// TwinCAT 3 PLC project Xplanar_First_Project
// ProgramVersion: 3.1.4023.0
// CompilerDefines: VISU_USEWSTRING
// libraries:
//   cyclic_database_recorder, * (Beckhoff K.K. - Japan)
//   JobManagementFramework, * (Bekchoff Automation K.K.)
//   Tc2_EtherCAT, * (Beckhoff Automation GmbH)
//   Tc2_Standard, * (Beckhoff Automation GmbH)
//   Tc2_System, * (Beckhoff Automation GmbH)
//   Tc2_Utilities, * (Beckhoff Automation GmbH)
//   Tc3_IotBase, * (Beckhoff Automation GmbH)
//   Tc3_JsonXml, * (Beckhoff Automation GmbH)
//   Tc3_Mc3PlanarMotion, * (Beckhoff Automation GmbH)
//   Tc3_Module, * (Beckhoff Automation GmbH)
//   Tc3_Physics, * (Beckhoff Automation GmbH)
//   Tc3_XPlanarUtility, * (Beckhoff Automation GmbH)
//   TwinCATDiagnosisTools, * (Beckhoff Automation K.K.)
//   VisuDialogs, * (System)
//   VisuSymbols,3.5.10.0,System
// project tree:
//   DUTs/ E_DbLogState.TcDUT (not stored), iManualCommand.TcDUT, JobEventReport.TcDUT, ManualCommand.TcDUT, sdo_xplanar_aps_diag.TcDUT, ST_database_aps_diag.TcDUT, ST_database_job_event.TcDUT, ST_mover_dynamics.TcDUT, ST_OperationPanel.TcDUT, ST_RouterStatusInfo.TcDUT, TileInfoType.TcDUT
//   / GlobalTextList.TcGTLO, PlcTask.TcTTO, RecipeManager.TcRMO (not stored), Visualization Manager.TcVMO (not stored)
//   GVLs/ GVL.TcGVL
//   POUs/ IoT.TcPOU, MAIN.TcPOU
//   POUs/model/activities/ FB_TaskMoveA_tilt_Creator.TcPOU, FB_TaskMoveB_tilt.TcPOU, FB_TaskMoveB_tilt_creator.TcPOU, FB_TaskMoveC_creator.TcPOU, FB_TaskMoveToPosition.TcPOU, FB_TaskMoveC.TcPOU, FB_TaskMoveToPosition_creator.TcPOU, FB_TaskMoveZ.TcPOU, FB_TaskMoveA_tilt.TcPOU, FB_TaskMoveZ_creator.TcPOU
//   POUs/model/IoT/ FB_JobReporter.TcPOU, FB_mqtt_publish.TcPOU, FB_serializer.TcPOU
//   VISUs/ ActionMode.TcTLO, MachineMode.TcTLO, Visualization.TcVIS, Visualization_operation.TcVIS, Visualization_recipe.TcVIS
// real-time tasks:
//   TASK Job Task: cycle default, priority 32
//   TASK MC-Task (MET): cycle T#2ms, priority 3, ADS port 521
//   TASK MC-Task (MPT): cycle T#10ms, priority 8, ADS port 531
//   TASK PlcTask: cycle T#10ms, priority 20, ADS port 352
//   TASK XPlanar Task3: cycle T#250us, priority 1, ADS port 350
// I/O:
//   DEVICE Device 3 (EtherCAT), AmsNetId 192.168.80.1.4.1
//     Term 1 (APS4322-7000) [APS4322-7000 Drive]
//       Term 2 (APS4322-5000) [APS4322-5000 Feedback]
//     Term 3 (APS4322-7000) [APS4322-7000 Drive]
//       Term 4 (APS4322-5000) [APS4322-5000 Feedback]
// variable links:
//   Device 3 (EtherCAT) <-> TcCOM Objects/XPlanar/Part1/Tile1
//     Term 3 (APS4322-7000)/APS Comm Inputs/CommStatusWord <-> Data Pointer/MoverCommStatusWord
//     Term 3 (APS4322-7000)/APS Comm Inputs/Data {1..4} <-> Data Pointer/MoverCommDataIn[{0..3}]  (4 links)
//     Term 3 (APS4322-7000)/APS Comm Outputs/CommControlWord <-> Data Pointer/MoverCommControlWord
//     Term 3 (APS4322-7000)/APS Comm Outputs/Data 1 <-> Data Pointer/MoverCommDataOut
//     Term 3 (APS4322-7000)/APS Diagdata/DC Link Voltage <-> Data Pointer/DcLinkVoltage
//     Term 3 (APS4322-7000)/APS Diagdata/Power supply current <-> Data Pointer/PowerSupplyCurrent
//     Term 3 (APS4322-7000)/APS Inputs/StatusWord <-> Data Pointer/PowerUnitStatusWord
//     Term 3 (APS4322-7000)/APS Outputs/ControlWord <-> Data Pointer/PowerUnitControlWord
//     Term 3 (APS4322-7000)/APS Outputs/Current D 0X0 <-> Data Pointer/DCurrentSetPoints[0]
//     Term 3 (APS4322-7000)/APS Outputs/Current D 0X1 <-> Data Pointer/DCurrentSetPoints[1]
//     Term 3 (APS4322-7000)/APS Outputs/Current D 0X2 <-> Data Pointer/DCurrentSetPoints[2]
//     Term 3 (APS4322-7000)/APS Outputs/Current D 1X0 <-> Data Pointer/DCurrentSetPoints[6]
//     Term 3 (APS4322-7000)/APS Outputs/Current D 1X1 <-> Data Pointer/DCurrentSetPoints[7]
//     Term 3 (APS4322-7000)/APS Outputs/Current D 1X2 <-> Data Pointer/DCurrentSetPoints[8]
//     Term 3 (APS4322-7000)/APS Outputs/Current D 2X0 <-> Data Pointer/DCurrentSetPoints[12]
//     Term 3 (APS4322-7000)/APS Outputs/Current D 2X1 <-> Data Pointer/DCurrentSetPoints[13]
//     Term 3 (APS4322-7000)/APS Outputs/Current D 2X2 <-> Data Pointer/DCurrentSetPoints[14]
//     Term 3 (APS4322-7000)/APS Outputs/Current D 3X0 <-> Data Pointer/DCurrentSetPoints[18]
//     Term 3 (APS4322-7000)/APS Outputs/Current D 3X1 <-> Data Pointer/DCurrentSetPoints[19]
//     Term 3 (APS4322-7000)/APS Outputs/Current D 3X2 <-> Data Pointer/DCurrentSetPoints[20]
//     Term 3 (APS4322-7000)/APS Outputs/Current D 0Y0 <-> Data Pointer/DCurrentSetPoints[3]
//     Term 3 (APS4322-7000)/APS Outputs/Current D 0Y1 <-> Data Pointer/DCurrentSetPoints[4]
//     Term 3 (APS4322-7000)/APS Outputs/Current D 0Y2 <-> Data Pointer/DCurrentSetPoints[5]
//     Term 3 (APS4322-7000)/APS Outputs/Current D 1Y0 <-> Data Pointer/DCurrentSetPoints[9]
//     Term 3 (APS4322-7000)/APS Outputs/Current D 1Y1 <-> Data Pointer/DCurrentSetPoints[10]
//     Term 3 (APS4322-7000)/APS Outputs/Current D 1Y2 <-> Data Pointer/DCurrentSetPoints[11]
//     Term 3 (APS4322-7000)/APS Outputs/Current D 2Y0 <-> Data Pointer/DCurrentSetPoints[15]
//     Term 3 (APS4322-7000)/APS Outputs/Current D 2Y1 <-> Data Pointer/DCurrentSetPoints[16]
//     Term 3 (APS4322-7000)/APS Outputs/Current D 2Y2 <-> Data Pointer/DCurrentSetPoints[17]
//     Term 3 (APS4322-7000)/APS Outputs/Current D 3Y0 <-> Data Pointer/DCurrentSetPoints[21]
//     Term 3 (APS4322-7000)/APS Outputs/Current D 3Y1 <-> Data Pointer/DCurrentSetPoints[22]
//     Term 3 (APS4322-7000)/APS Outputs/Current D 3Y2 <-> Data Pointer/DCurrentSetPoints[23]
//     Term 3 (APS4322-7000)/APS Outputs/Current Q 0X0 <-> Data Pointer/QCurrentSetPoints[0]
//     Term 3 (APS4322-7000)/APS Outputs/Current Q 0X1 <-> Data Pointer/QCurrentSetPoints[1]
//     Term 3 (APS4322-7000)/APS Outputs/Current Q 0X2 <-> Data Pointer/QCurrentSetPoints[2]
//     Term 3 (APS4322-7000)/APS Outputs/Current Q 1X0 <-> Data Pointer/QCurrentSetPoints[6]
//     Term 3 (APS4322-7000)/APS Outputs/Current Q 1X1 <-> Data Pointer/QCurrentSetPoints[7]
//     Term 3 (APS4322-7000)/APS Outputs/Current Q 1X2 <-> Data Pointer/QCurrentSetPoints[8]
//     Term 3 (APS4322-7000)/APS Outputs/Current Q 2X0 <-> Data Pointer/QCurrentSetPoints[12]
//     Term 3 (APS4322-7000)/APS Outputs/Current Q 2X1 <-> Data Pointer/QCurrentSetPoints[13]
//     Term 3 (APS4322-7000)/APS Outputs/Current Q 2X2 <-> Data Pointer/QCurrentSetPoints[14]
//     Term 3 (APS4322-7000)/APS Outputs/Current Q 3X0 <-> Data Pointer/QCurrentSetPoints[18]
//     Term 3 (APS4322-7000)/APS Outputs/Current Q 3X1 <-> Data Pointer/QCurrentSetPoints[19]
//     Term 3 (APS4322-7000)/APS Outputs/Current Q 3X2 <-> Data Pointer/QCurrentSetPoints[20]
//     Term 3 (APS4322-7000)/APS Outputs/Current Q 0Y0 <-> Data Pointer/QCurrentSetPoints[3]
//     Term 3 (APS4322-7000)/APS Outputs/Current Q 0Y1 <-> Data Pointer/QCurrentSetPoints[4]
//     Term 3 (APS4322-7000)/APS Outputs/Current Q 0Y2 <-> Data Pointer/QCurrentSetPoints[5]
//     Term 3 (APS4322-7000)/APS Outputs/Current Q 1Y0 <-> Data Pointer/QCurrentSetPoints[9]
//     Term 3 (APS4322-7000)/APS Outputs/Current Q 1Y1 <-> Data Pointer/QCurrentSetPoints[10]
//     Term 3 (APS4322-7000)/APS Outputs/Current Q 1Y2 <-> Data Pointer/QCurrentSetPoints[11]
//     Term 3 (APS4322-7000)/APS Outputs/Current Q 2Y0 <-> Data Pointer/QCurrentSetPoints[15]
//     Term 3 (APS4322-7000)/APS Outputs/Current Q 2Y1 <-> Data Pointer/QCurrentSetPoints[16]
//     Term 3 (APS4322-7000)/APS Outputs/Current Q 2Y2 <-> Data Pointer/QCurrentSetPoints[17]
//     Term 3 (APS4322-7000)/APS Outputs/Current Q 3Y0 <-> Data Pointer/QCurrentSetPoints[21]
//     Term 3 (APS4322-7000)/APS Outputs/Current Q 3Y1 <-> Data Pointer/QCurrentSetPoints[22]
//     Term 3 (APS4322-7000)/APS Outputs/Current Q 3Y2 <-> Data Pointer/QCurrentSetPoints[23]
//     Term 3 (APS4322-7000)/APS Outputs/PhiE 0X0 <-> Data Pointer/PhiSetPoints[0]
//     Term 3 (APS4322-7000)/APS Outputs/PhiE 0X1 <-> Data Pointer/PhiSetPoints[1]
//     Term 3 (APS4322-7000)/APS Outputs/PhiE 0X2 <-> Data Pointer/PhiSetPoints[2]
//     Term 3 (APS4322-7000)/APS Outputs/PhiE 1X0 <-> Data Pointer/PhiSetPoints[6]
//     Term 3 (APS4322-7000)/APS Outputs/PhiE 1X1 <-> Data Pointer/PhiSetPoints[7]
//     Term 3 (APS4322-7000)/APS Outputs/PhiE 1X2 <-> Data Pointer/PhiSetPoints[8]
//     Term 3 (APS4322-7000)/APS Outputs/PhiE 2X0 <-> Data Pointer/PhiSetPoints[12]
//     Term 3 (APS4322-7000)/APS Outputs/PhiE 2X1 <-> Data Pointer/PhiSetPoints[13]
//     Term 3 (APS4322-7000)/APS Outputs/PhiE 2X2 <-> Data Pointer/PhiSetPoints[14]
//     Term 3 (APS4322-7000)/APS Outputs/PhiE 3X0 <-> Data Pointer/PhiSetPoints[18]
//     Term 3 (APS4322-7000)/APS Outputs/PhiE 3X1 <-> Data Pointer/PhiSetPoints[19]
//     Term 3 (APS4322-7000)/APS Outputs/PhiE 3X2 <-> Data Pointer/PhiSetPoints[20]
//     Term 3 (APS4322-7000)/APS Outputs/PhiE 0Y0 <-> Data Pointer/PhiSetPoints[3]
//     Term 3 (APS4322-7000)/APS Outputs/PhiE 0Y1 <-> Data Pointer/PhiSetPoints[4]
//     Term 3 (APS4322-7000)/APS Outputs/PhiE 0Y2 <-> Data Pointer/PhiSetPoints[5]
//     Term 3 (APS4322-7000)/APS Outputs/PhiE 1Y0 <-> Data Pointer/PhiSetPoints[9]
//     Term 3 (APS4322-7000)/APS Outputs/PhiE 1Y1 <-> Data Pointer/PhiSetPoints[10]
//     Term 3 (APS4322-7000)/APS Outputs/PhiE 1Y2 <-> Data Pointer/PhiSetPoints[11]
//     Term 3 (APS4322-7000)/APS Outputs/PhiE 2Y0 <-> Data Pointer/PhiSetPoints[15]
//     Term 3 (APS4322-7000)/APS Outputs/PhiE 2Y1 <-> Data Pointer/PhiSetPoints[16]
//     Term 3 (APS4322-7000)/APS Outputs/PhiE 2Y2 <-> Data Pointer/PhiSetPoints[17]
//     Term 3 (APS4322-7000)/APS Outputs/PhiE 3Y0 <-> Data Pointer/PhiSetPoints[21]
//     Term 3 (APS4322-7000)/APS Outputs/PhiE 3Y1 <-> Data Pointer/PhiSetPoints[22]
//     Term 3 (APS4322-7000)/APS Outputs/PhiE 3Y2 <-> Data Pointer/PhiSetPoints[23]
//     Term 3 (APS4322-7000)/Term 4 (APS4322-5000)/FB Inputs/A{0..8 step 2} X-Field <-> Data Pointer/HallSensorFieldsXYZ[{0..12 step 3}]  (5 links)
//     Term 3 (APS4322-7000)/Term 4 (APS4322-5000)/FB Inputs/A{0..8 step 2} Y-Field <-> Data Pointer/HallSensorFieldsXYZ[{1..13 step 3}]  (5 links)
//     Term 3 (APS4322-7000)/Term 4 (APS4322-5000)/FB Inputs/A{0..8 step 2} Z-Field <-> Data Pointer/HallSensorFieldsXYZ[{2..14 step 3}]  (5 links)
//     Term 3 (APS4322-7000)/Term 4 (APS4322-5000)/FB Inputs/B{1..9 step 2} X-Field <-> Data Pointer/HallSensorFieldsXYZ[{15..27 step 3}]  (5 links)
//     Term 3 (APS4322-7000)/Term 4 (APS4322-5000)/FB Inputs/B{1..9 step 2} Y-Field <-> Data Pointer/HallSensorFieldsXYZ[{16..28 step 3}]  (5 links)
//     Term 3 (APS4322-7000)/Term 4 (APS4322-5000)/FB Inputs/B{1..9 step 2} Z-Field <-> Data Pointer/HallSensorFieldsXYZ[{17..29 step 3}]  (5 links)
//     Term 3 (APS4322-7000)/Term 4 (APS4322-5000)/FB Inputs/C{0..8 step 2} X-Field <-> Data Pointer/HallSensorFieldsXYZ[{30..42 step 3}]  (5 links)
//     Term 3 (APS4322-7000)/Term 4 (APS4322-5000)/FB Inputs/C{0..8 step 2} Y-Field <-> Data Pointer/HallSensorFieldsXYZ[{31..43 step 3}]  (5 links)
//     Term 3 (APS4322-7000)/Term 4 (APS4322-5000)/FB Inputs/C{0..8 step 2} Z-Field <-> Data Pointer/HallSensorFieldsXYZ[{32..44 step 3}]  (5 links)
//     Term 3 (APS4322-7000)/Term 4 (APS4322-5000)/FB Inputs/D{1..9 step 2} X-Field <-> Data Pointer/HallSensorFieldsXYZ[{45..57 step 3}]  (5 links)
//     Term 3 (APS4322-7000)/Term 4 (APS4322-5000)/FB Inputs/D{1..9 step 2} Y-Field <-> Data Pointer/HallSensorFieldsXYZ[{46..58 step 3}]  (5 links)
//     Term 3 (APS4322-7000)/Term 4 (APS4322-5000)/FB Inputs/D{1..9 step 2} Z-Field <-> Data Pointer/HallSensorFieldsXYZ[{47..59 step 3}]  (5 links)
//     Term 3 (APS4322-7000)/Term 4 (APS4322-5000)/FB Inputs/E{0..8 step 2} X-Field <-> Data Pointer/HallSensorFieldsXYZ[{60..72 step 3}]  (5 links)
//     Term 3 (APS4322-7000)/Term 4 (APS4322-5000)/FB Inputs/E{0..8 step 2} Y-Field <-> Data Pointer/HallSensorFieldsXYZ[{61..73 step 3}]  (5 links)
//     Term 3 (APS4322-7000)/Term 4 (APS4322-5000)/FB Inputs/E{0..8 step 2} Z-Field <-> Data Pointer/HallSensorFieldsXYZ[{62..74 step 3}]  (5 links)
//     Term 3 (APS4322-7000)/Term 4 (APS4322-5000)/FB Inputs/F{1..9 step 2} X-Field <-> Data Pointer/HallSensorFieldsXYZ[{75..87 step 3}]  (5 links)
//     Term 3 (APS4322-7000)/Term 4 (APS4322-5000)/FB Inputs/F{1..9 step 2} Y-Field <-> Data Pointer/HallSensorFieldsXYZ[{76..88 step 3}]  (5 links)
//     Term 3 (APS4322-7000)/Term 4 (APS4322-5000)/FB Inputs/F{1..9 step 2} Z-Field <-> Data Pointer/HallSensorFieldsXYZ[{77..89 step 3}]  (5 links)
//     Term 3 (APS4322-7000)/Term 4 (APS4322-5000)/FB Inputs/G{0..8 step 2} X-Field <-> Data Pointer/HallSensorFieldsXYZ[{90..102 step 3}]  (5 links)
//     Term 3 (APS4322-7000)/Term 4 (APS4322-5000)/FB Inputs/G{0..8 step 2} Y-Field <-> Data Pointer/HallSensorFieldsXYZ[{91..103 step 3}]  (5 links)
//     Term 3 (APS4322-7000)/Term 4 (APS4322-5000)/FB Inputs/G{0..8 step 2} Z-Field <-> Data Pointer/HallSensorFieldsXYZ[{92..104 step 3}]  (5 links)
//     Term 3 (APS4322-7000)/Term 4 (APS4322-5000)/FB Inputs/H{1..9 step 2} X-Field <-> Data Pointer/HallSensorFieldsXYZ[{105..117 step 3}]  (5 links)
//     Term 3 (APS4322-7000)/Term 4 (APS4322-5000)/FB Inputs/H{1..9 step 2} Y-Field <-> Data Pointer/HallSensorFieldsXYZ[{106..118 step 3}]  (5 links)
//     Term 3 (APS4322-7000)/Term 4 (APS4322-5000)/FB Inputs/H{1..9 step 2} Z-Field <-> Data Pointer/HallSensorFieldsXYZ[{107..119 step 3}]  (5 links)
//     Term 3 (APS4322-7000)/Term 4 (APS4322-5000)/FB Inputs/I{0..8 step 2} X-Field <-> Data Pointer/HallSensorFieldsXYZ[{120..132 step 3}]  (5 links)
//     Term 3 (APS4322-7000)/Term 4 (APS4322-5000)/FB Inputs/I{0..8 step 2} Y-Field <-> Data Pointer/HallSensorFieldsXYZ[{121..133 step 3}]  (5 links)
//     Term 3 (APS4322-7000)/Term 4 (APS4322-5000)/FB Inputs/I{0..8 step 2} Z-Field <-> Data Pointer/HallSensorFieldsXYZ[{122..134 step 3}]  (5 links)
//     Term 3 (APS4322-7000)/Term 4 (APS4322-5000)/FB Inputs/J{1..9 step 2} X-Field <-> Data Pointer/HallSensorFieldsXYZ[{135..147 step 3}]  (5 links)
//     Term 3 (APS4322-7000)/Term 4 (APS4322-5000)/FB Inputs/J{1..9 step 2} Y-Field <-> Data Pointer/HallSensorFieldsXYZ[{136..148 step 3}]  (5 links)
//     Term 3 (APS4322-7000)/Term 4 (APS4322-5000)/FB Inputs/J{1..9 step 2} Z-Field <-> Data Pointer/HallSensorFieldsXYZ[{137..149 step 3}]  (5 links)
//     Term 3 (APS4322-7000)/Term 4 (APS4322-5000)/FB Inputs/Status <-> Data Pointer/FeedbackStatus
//   Device 3 (EtherCAT) <-> TcCOM Objects/XPlanar/Part1/Tile2
//     Term 1 (APS4322-7000)/APS Comm Inputs/CommStatusWord <-> Data Pointer/MoverCommStatusWord
//     Term 1 (APS4322-7000)/APS Comm Inputs/Data {1..4} <-> Data Pointer/MoverCommDataIn[{0..3}]  (4 links)
//     Term 1 (APS4322-7000)/APS Comm Outputs/CommControlWord <-> Data Pointer/MoverCommControlWord
//     Term 1 (APS4322-7000)/APS Comm Outputs/Data 1 <-> Data Pointer/MoverCommDataOut
//     Term 1 (APS4322-7000)/APS Diagdata/DC Link Voltage <-> Data Pointer/DcLinkVoltage
//     Term 1 (APS4322-7000)/APS Diagdata/Power supply current <-> Data Pointer/PowerSupplyCurrent
//     Term 1 (APS4322-7000)/APS Inputs/StatusWord <-> Data Pointer/PowerUnitStatusWord
//     Term 1 (APS4322-7000)/APS Outputs/ControlWord <-> Data Pointer/PowerUnitControlWord
//     Term 1 (APS4322-7000)/APS Outputs/Current D 0X0 <-> Data Pointer/DCurrentSetPoints[0]
//     Term 1 (APS4322-7000)/APS Outputs/Current D 0X1 <-> Data Pointer/DCurrentSetPoints[1]
//     Term 1 (APS4322-7000)/APS Outputs/Current D 0X2 <-> Data Pointer/DCurrentSetPoints[2]
//     Term 1 (APS4322-7000)/APS Outputs/Current D 1X0 <-> Data Pointer/DCurrentSetPoints[6]
//     Term 1 (APS4322-7000)/APS Outputs/Current D 1X1 <-> Data Pointer/DCurrentSetPoints[7]
//     Term 1 (APS4322-7000)/APS Outputs/Current D 1X2 <-> Data Pointer/DCurrentSetPoints[8]
//     Term 1 (APS4322-7000)/APS Outputs/Current D 2X0 <-> Data Pointer/DCurrentSetPoints[12]
//     Term 1 (APS4322-7000)/APS Outputs/Current D 2X1 <-> Data Pointer/DCurrentSetPoints[13]
//     Term 1 (APS4322-7000)/APS Outputs/Current D 2X2 <-> Data Pointer/DCurrentSetPoints[14]
//     Term 1 (APS4322-7000)/APS Outputs/Current D 3X0 <-> Data Pointer/DCurrentSetPoints[18]
//     Term 1 (APS4322-7000)/APS Outputs/Current D 3X1 <-> Data Pointer/DCurrentSetPoints[19]
//     Term 1 (APS4322-7000)/APS Outputs/Current D 3X2 <-> Data Pointer/DCurrentSetPoints[20]
//     Term 1 (APS4322-7000)/APS Outputs/Current D 0Y0 <-> Data Pointer/DCurrentSetPoints[3]
//     Term 1 (APS4322-7000)/APS Outputs/Current D 0Y1 <-> Data Pointer/DCurrentSetPoints[4]
//     Term 1 (APS4322-7000)/APS Outputs/Current D 0Y2 <-> Data Pointer/DCurrentSetPoints[5]
//     Term 1 (APS4322-7000)/APS Outputs/Current D 1Y0 <-> Data Pointer/DCurrentSetPoints[9]
//     Term 1 (APS4322-7000)/APS Outputs/Current D 1Y1 <-> Data Pointer/DCurrentSetPoints[10]
//     Term 1 (APS4322-7000)/APS Outputs/Current D 1Y2 <-> Data Pointer/DCurrentSetPoints[11]
//     Term 1 (APS4322-7000)/APS Outputs/Current D 2Y0 <-> Data Pointer/DCurrentSetPoints[15]
//     Term 1 (APS4322-7000)/APS Outputs/Current D 2Y1 <-> Data Pointer/DCurrentSetPoints[16]
//     Term 1 (APS4322-7000)/APS Outputs/Current D 2Y2 <-> Data Pointer/DCurrentSetPoints[17]
//     Term 1 (APS4322-7000)/APS Outputs/Current D 3Y0 <-> Data Pointer/DCurrentSetPoints[21]
//     Term 1 (APS4322-7000)/APS Outputs/Current D 3Y1 <-> Data Pointer/DCurrentSetPoints[22]
//     Term 1 (APS4322-7000)/APS Outputs/Current D 3Y2 <-> Data Pointer/DCurrentSetPoints[23]
//     Term 1 (APS4322-7000)/APS Outputs/Current Q 0X0 <-> Data Pointer/QCurrentSetPoints[0]
//     Term 1 (APS4322-7000)/APS Outputs/Current Q 0X1 <-> Data Pointer/QCurrentSetPoints[1]
//     Term 1 (APS4322-7000)/APS Outputs/Current Q 0X2 <-> Data Pointer/QCurrentSetPoints[2]
//     Term 1 (APS4322-7000)/APS Outputs/Current Q 1X0 <-> Data Pointer/QCurrentSetPoints[6]
//     Term 1 (APS4322-7000)/APS Outputs/Current Q 1X1 <-> Data Pointer/QCurrentSetPoints[7]
//     Term 1 (APS4322-7000)/APS Outputs/Current Q 1X2 <-> Data Pointer/QCurrentSetPoints[8]
//     Term 1 (APS4322-7000)/APS Outputs/Current Q 2X0 <-> Data Pointer/QCurrentSetPoints[12]
//     Term 1 (APS4322-7000)/APS Outputs/Current Q 2X1 <-> Data Pointer/QCurrentSetPoints[13]
//     Term 1 (APS4322-7000)/APS Outputs/Current Q 2X2 <-> Data Pointer/QCurrentSetPoints[14]
//     Term 1 (APS4322-7000)/APS Outputs/Current Q 3X0 <-> Data Pointer/QCurrentSetPoints[18]
//     Term 1 (APS4322-7000)/APS Outputs/Current Q 3X1 <-> Data Pointer/QCurrentSetPoints[19]
//     Term 1 (APS4322-7000)/APS Outputs/Current Q 3X2 <-> Data Pointer/QCurrentSetPoints[20]
//     Term 1 (APS4322-7000)/APS Outputs/Current Q 0Y0 <-> Data Pointer/QCurrentSetPoints[3]
//     Term 1 (APS4322-7000)/APS Outputs/Current Q 0Y1 <-> Data Pointer/QCurrentSetPoints[4]
//     Term 1 (APS4322-7000)/APS Outputs/Current Q 0Y2 <-> Data Pointer/QCurrentSetPoints[5]
//     Term 1 (APS4322-7000)/APS Outputs/Current Q 1Y0 <-> Data Pointer/QCurrentSetPoints[9]
//     Term 1 (APS4322-7000)/APS Outputs/Current Q 1Y1 <-> Data Pointer/QCurrentSetPoints[10]
//     Term 1 (APS4322-7000)/APS Outputs/Current Q 1Y2 <-> Data Pointer/QCurrentSetPoints[11]
//     Term 1 (APS4322-7000)/APS Outputs/Current Q 2Y0 <-> Data Pointer/QCurrentSetPoints[15]
//     Term 1 (APS4322-7000)/APS Outputs/Current Q 2Y1 <-> Data Pointer/QCurrentSetPoints[16]
//     Term 1 (APS4322-7000)/APS Outputs/Current Q 2Y2 <-> Data Pointer/QCurrentSetPoints[17]
//     Term 1 (APS4322-7000)/APS Outputs/Current Q 3Y0 <-> Data Pointer/QCurrentSetPoints[21]
//     Term 1 (APS4322-7000)/APS Outputs/Current Q 3Y1 <-> Data Pointer/QCurrentSetPoints[22]
//     Term 1 (APS4322-7000)/APS Outputs/Current Q 3Y2 <-> Data Pointer/QCurrentSetPoints[23]
//     Term 1 (APS4322-7000)/APS Outputs/PhiE 0X0 <-> Data Pointer/PhiSetPoints[0]
//     Term 1 (APS4322-7000)/APS Outputs/PhiE 0X1 <-> Data Pointer/PhiSetPoints[1]
//     Term 1 (APS4322-7000)/APS Outputs/PhiE 0X2 <-> Data Pointer/PhiSetPoints[2]
//     Term 1 (APS4322-7000)/APS Outputs/PhiE 1X0 <-> Data Pointer/PhiSetPoints[6]
//     Term 1 (APS4322-7000)/APS Outputs/PhiE 1X1 <-> Data Pointer/PhiSetPoints[7]
//     Term 1 (APS4322-7000)/APS Outputs/PhiE 1X2 <-> Data Pointer/PhiSetPoints[8]
//     Term 1 (APS4322-7000)/APS Outputs/PhiE 2X0 <-> Data Pointer/PhiSetPoints[12]
//     Term 1 (APS4322-7000)/APS Outputs/PhiE 2X1 <-> Data Pointer/PhiSetPoints[13]
//     Term 1 (APS4322-7000)/APS Outputs/PhiE 2X2 <-> Data Pointer/PhiSetPoints[14]
//     Term 1 (APS4322-7000)/APS Outputs/PhiE 3X0 <-> Data Pointer/PhiSetPoints[18]
//     Term 1 (APS4322-7000)/APS Outputs/PhiE 3X1 <-> Data Pointer/PhiSetPoints[19]
//     Term 1 (APS4322-7000)/APS Outputs/PhiE 3X2 <-> Data Pointer/PhiSetPoints[20]
//     Term 1 (APS4322-7000)/APS Outputs/PhiE 0Y0 <-> Data Pointer/PhiSetPoints[3]
//     Term 1 (APS4322-7000)/APS Outputs/PhiE 0Y1 <-> Data Pointer/PhiSetPoints[4]
//     Term 1 (APS4322-7000)/APS Outputs/PhiE 0Y2 <-> Data Pointer/PhiSetPoints[5]
//     Term 1 (APS4322-7000)/APS Outputs/PhiE 1Y0 <-> Data Pointer/PhiSetPoints[9]
//     Term 1 (APS4322-7000)/APS Outputs/PhiE 1Y1 <-> Data Pointer/PhiSetPoints[10]
//     Term 1 (APS4322-7000)/APS Outputs/PhiE 1Y2 <-> Data Pointer/PhiSetPoints[11]
//     Term 1 (APS4322-7000)/APS Outputs/PhiE 2Y0 <-> Data Pointer/PhiSetPoints[15]
//     Term 1 (APS4322-7000)/APS Outputs/PhiE 2Y1 <-> Data Pointer/PhiSetPoints[16]
//     Term 1 (APS4322-7000)/APS Outputs/PhiE 2Y2 <-> Data Pointer/PhiSetPoints[17]
//     Term 1 (APS4322-7000)/APS Outputs/PhiE 3Y0 <-> Data Pointer/PhiSetPoints[21]
//     Term 1 (APS4322-7000)/APS Outputs/PhiE 3Y1 <-> Data Pointer/PhiSetPoints[22]
//     Term 1 (APS4322-7000)/APS Outputs/PhiE 3Y2 <-> Data Pointer/PhiSetPoints[23]
//     Term 1 (APS4322-7000)/Term 2 (APS4322-5000)/FB Inputs/A{0..8 step 2} X-Field <-> Data Pointer/HallSensorFieldsXYZ[{0..12 step 3}]  (5 links)
//     Term 1 (APS4322-7000)/Term 2 (APS4322-5000)/FB Inputs/A{0..8 step 2} Y-Field <-> Data Pointer/HallSensorFieldsXYZ[{1..13 step 3}]  (5 links)
//     Term 1 (APS4322-7000)/Term 2 (APS4322-5000)/FB Inputs/A{0..8 step 2} Z-Field <-> Data Pointer/HallSensorFieldsXYZ[{2..14 step 3}]  (5 links)
//     Term 1 (APS4322-7000)/Term 2 (APS4322-5000)/FB Inputs/B{1..9 step 2} X-Field <-> Data Pointer/HallSensorFieldsXYZ[{15..27 step 3}]  (5 links)
//     Term 1 (APS4322-7000)/Term 2 (APS4322-5000)/FB Inputs/B{1..9 step 2} Y-Field <-> Data Pointer/HallSensorFieldsXYZ[{16..28 step 3}]  (5 links)
//     Term 1 (APS4322-7000)/Term 2 (APS4322-5000)/FB Inputs/B{1..9 step 2} Z-Field <-> Data Pointer/HallSensorFieldsXYZ[{17..29 step 3}]  (5 links)
//     Term 1 (APS4322-7000)/Term 2 (APS4322-5000)/FB Inputs/C{0..8 step 2} X-Field <-> Data Pointer/HallSensorFieldsXYZ[{30..42 step 3}]  (5 links)
//     Term 1 (APS4322-7000)/Term 2 (APS4322-5000)/FB Inputs/C{0..8 step 2} Y-Field <-> Data Pointer/HallSensorFieldsXYZ[{31..43 step 3}]  (5 links)
//     Term 1 (APS4322-7000)/Term 2 (APS4322-5000)/FB Inputs/C{0..8 step 2} Z-Field <-> Data Pointer/HallSensorFieldsXYZ[{32..44 step 3}]  (5 links)
//     Term 1 (APS4322-7000)/Term 2 (APS4322-5000)/FB Inputs/D{1..9 step 2} X-Field <-> Data Pointer/HallSensorFieldsXYZ[{45..57 step 3}]  (5 links)
//     Term 1 (APS4322-7000)/Term 2 (APS4322-5000)/FB Inputs/D{1..9 step 2} Y-Field <-> Data Pointer/HallSensorFieldsXYZ[{46..58 step 3}]  (5 links)
//     Term 1 (APS4322-7000)/Term 2 (APS4322-5000)/FB Inputs/D{1..9 step 2} Z-Field <-> Data Pointer/HallSensorFieldsXYZ[{47..59 step 3}]  (5 links)
//     Term 1 (APS4322-7000)/Term 2 (APS4322-5000)/FB Inputs/E{0..8 step 2} X-Field <-> Data Pointer/HallSensorFieldsXYZ[{60..72 step 3}]  (5 links)
//     Term 1 (APS4322-7000)/Term 2 (APS4322-5000)/FB Inputs/E{0..8 step 2} Y-Field <-> Data Pointer/HallSensorFieldsXYZ[{61..73 step 3}]  (5 links)
//     Term 1 (APS4322-7000)/Term 2 (APS4322-5000)/FB Inputs/E{0..8 step 2} Z-Field <-> Data Pointer/HallSensorFieldsXYZ[{62..74 step 3}]  (5 links)
//     Term 1 (APS4322-7000)/Term 2 (APS4322-5000)/FB Inputs/F{1..9 step 2} X-Field <-> Data Pointer/HallSensorFieldsXYZ[{75..87 step 3}]  (5 links)
//     Term 1 (APS4322-7000)/Term 2 (APS4322-5000)/FB Inputs/F{1..9 step 2} Y-Field <-> Data Pointer/HallSensorFieldsXYZ[{76..88 step 3}]  (5 links)
//     Term 1 (APS4322-7000)/Term 2 (APS4322-5000)/FB Inputs/F{1..9 step 2} Z-Field <-> Data Pointer/HallSensorFieldsXYZ[{77..89 step 3}]  (5 links)
//     Term 1 (APS4322-7000)/Term 2 (APS4322-5000)/FB Inputs/G{0..8 step 2} X-Field <-> Data Pointer/HallSensorFieldsXYZ[{90..102 step 3}]  (5 links)
//     Term 1 (APS4322-7000)/Term 2 (APS4322-5000)/FB Inputs/G{0..8 step 2} Y-Field <-> Data Pointer/HallSensorFieldsXYZ[{91..103 step 3}]  (5 links)
//     Term 1 (APS4322-7000)/Term 2 (APS4322-5000)/FB Inputs/G{0..8 step 2} Z-Field <-> Data Pointer/HallSensorFieldsXYZ[{92..104 step 3}]  (5 links)
//     Term 1 (APS4322-7000)/Term 2 (APS4322-5000)/FB Inputs/H{1..9 step 2} X-Field <-> Data Pointer/HallSensorFieldsXYZ[{105..117 step 3}]  (5 links)
//     Term 1 (APS4322-7000)/Term 2 (APS4322-5000)/FB Inputs/H{1..9 step 2} Y-Field <-> Data Pointer/HallSensorFieldsXYZ[{106..118 step 3}]  (5 links)
//     Term 1 (APS4322-7000)/Term 2 (APS4322-5000)/FB Inputs/H{1..9 step 2} Z-Field <-> Data Pointer/HallSensorFieldsXYZ[{107..119 step 3}]  (5 links)
//     Term 1 (APS4322-7000)/Term 2 (APS4322-5000)/FB Inputs/I{0..8 step 2} X-Field <-> Data Pointer/HallSensorFieldsXYZ[{120..132 step 3}]  (5 links)
//     Term 1 (APS4322-7000)/Term 2 (APS4322-5000)/FB Inputs/I{0..8 step 2} Y-Field <-> Data Pointer/HallSensorFieldsXYZ[{121..133 step 3}]  (5 links)
//     Term 1 (APS4322-7000)/Term 2 (APS4322-5000)/FB Inputs/I{0..8 step 2} Z-Field <-> Data Pointer/HallSensorFieldsXYZ[{122..134 step 3}]  (5 links)
//     Term 1 (APS4322-7000)/Term 2 (APS4322-5000)/FB Inputs/J{1..9 step 2} X-Field <-> Data Pointer/HallSensorFieldsXYZ[{135..147 step 3}]  (5 links)
//     Term 1 (APS4322-7000)/Term 2 (APS4322-5000)/FB Inputs/J{1..9 step 2} Y-Field <-> Data Pointer/HallSensorFieldsXYZ[{136..148 step 3}]  (5 links)
//     Term 1 (APS4322-7000)/Term 2 (APS4322-5000)/FB Inputs/J{1..9 step 2} Z-Field <-> Data Pointer/HallSensorFieldsXYZ[{137..149 step 3}]  (5 links)
//     Term 1 (APS4322-7000)/Term 2 (APS4322-5000)/FB Inputs/Status <-> Data Pointer/FeedbackStatus
//   XPlanar MC Project/Axes/Mover4220_1 <-> TcCOM Objects/XPlanar/Mover4220_1
//     McToIo/STD <-> InputsFromNC3/NC3ToHW
//   Xplanar_First_Project/Xplanar_First_Project Instance <-> XPlanar MC Project/Axes/Mover4220_1
//     PlcTask Inputs/GVL.planar_movers[1].MCTOPLC/ACT <-> McToPlc/ACT
//     PlcTask Inputs/GVL.planar_movers[1].MCTOPLC/COORDMODE <-> McToPlc/COORDMODE
//     PlcTask Inputs/GVL.planar_movers[1].MCTOPLC/SET <-> McToPlc/SET
//     PlcTask Inputs/GVL.planar_movers[1].MCTOPLC/SETONTRACK <-> McToPlc/SETONTRACK
//     PlcTask Inputs/GVL.planar_movers[1].MCTOPLC/STD <-> McToPlc/STD
//     PlcTask Outputs/GVL.planar_movers[1].PLCTOMC/STD <-> PlcToMc/STD
//   TcCOM Objects/XPlanar/Mover4220_1 <-> XPlanar MC Project/Axes/Mover4220_1
//     OutputsToNC3/HWToNC3 <-> IoToMc/STD

CONFIGURATION Xplanar_First_Project
    RESOURCE PLC ON TwinCAT3
        TASK PlcTask(INTERVAL := T#10ms, PRIORITY := 20);
        PROGRAM MAIN WITH PlcTask : MAIN;
    END_RESOURCE
END_CONFIGURATION

// ---- DUTs/iManualCommand.TcDUT
TYPE iManualCommand :
UNION
	i_com: UINT;
	com: ManualCommand;
END_UNION
END_TYPE

// ---- DUTs/JobEventReport.TcDUT
{attribute ‘pack_mode’ := ‘1’}
TYPE JobEventReport :
STRUCT
	old_state	: STRING;
	new_state	: STRING;
	record_time	: STRING;
	{attribute 'TcEncoding':='UTF-8'}
	job_id		: STRING;
	{attribute 'TcEncoding':='UTF-8'}
	task_name	: STRING;
	erro_id		: UDINT;
END_STRUCT
END_TYPE

// ---- DUTs/ManualCommand.TcDUT
{attribute 'qualified_only'}
{attribute 'strict'}
TYPE ManualCommand :
(
	move_pos_L1 := 0,
	move_pos_L2,
	move_pos_L3,
	move_pos_c1,
	move_pos_c2,
	move_pos_c3,
	move_pos_r1,
	move_pos_r2,
	move_pos_r3,
	move_up,
	move_down,
	move_tilt_up_front,
	move_tilt_up_rear,
	move_tilt_up_right,
	move_tilt_up_left,
	move_tilt_horizontal,
	move_roll_w,
	move_roll_n,
	move_roll_e,
	move_roll_s
);
END_TYPE

// ---- DUTs/sdo_xplanar_aps_diag.TcDUT
{attribute 'TcAnalytics'}
{attribute 'pack_mode' := '4'}
TYPE sdo_xplanar_aps_diag :
STRUCT
  identity: USINT;
  {attribute 'FieldName' := 'dc_link_voltage'}
  dc_link_voltage: DINT;
  {attribute 'FieldName' := 'power_supply_current'}
  power_supply_current: DINT;
  {attribute 'FieldName' := 'temperature_north'}
  temperature_north: UINT;
  {attribute 'FieldName' := 'temperature_east'}
  temperature_east: UINT;
  {attribute 'FieldName' := 'temperature_south'}
  temperature_south: UINT;
  {attribute 'FieldName' := 'temperature_west'}
  temperature_west: UINT;
  {attribute 'FieldName' := 'temperature_center'}
  temperature_center: UINT;
  {attribute 'FieldName' := 'temperature_power'}
  temperature_power: UINT;
  {attribute 'FieldName' := 'fan_rpm'}
  fan_rpm: UINT;
  {attribute 'FieldName' := 'fan_duty_cycle'}
  fan_duty_cycle: USINT;
  {attribute 'FieldName' := 'supply_voltage_us'}
  supply_voltage_us: UDINT;
  {attribute 'FieldName' := 'auxiliary_voltage'}
  auxiliary_voltage: UDINT;
  {attribute 'FieldName' := 'acceleration_x'}
  acceleration_x: UDINT;
  {attribute 'FieldName' := 'acceleration_y'}
  acceleration_y: UDINT;
  {attribute 'FieldName' := 'acceleration_z'}
  acceleration_z: UDINT;
  {attribute 'FieldName' := 'time_to_shutdown'}
  time_to_shutdown: UDINT;
  {attribute 'FieldName' := 'fb_fw_rev'}
  fb_fw_rev: UDINT;
END_STRUCT
END_TYPE

// ---- DUTs/ST_database_aps_diag.TcDUT
{attribute 'pack_mode' := '1'}
TYPE ST_database_aps_diag:
STRUCT
	{attribute 'TagName' := 'tile_number'}
	tile_number :STRING;
	{attribute 'FieldName' := 'dc_link_voltage'}
	dc_link_voltage: DINT;
	{attribute 'FieldName' := 'power_supply_current'}
	power_supply_current: DINT;
	{attribute 'FieldName' := 'temperature_north'}
	temperature_north: DINT;
	{attribute 'FieldName' := 'temperature_east'}
	temperature_east: DINT;
	{attribute 'FieldName' := 'temperature_south'}
	temperature_south: DINT;
	{attribute 'FieldName' := 'temperature_west'}
	temperature_west: DINT;
	{attribute 'FieldName' := 'temperature_center'}
	temperature_center: DINT;
	{attribute 'FieldName' := 'temperature_power'}
	temperature_power: DINT;
	{attribute 'FieldName' := 'fan_rpm'}
	fan_rpm: DINT;
	{attribute 'FieldName' := 'fan_duty_cycle'}
	fan_duty_cycle: INT;
	{attribute 'FieldName' := 'supply_voltage_us'}
	supply_voltage_us: LINT;
	{attribute 'FieldName' := 'auxiliary_voltage'}
	auxiliary_voltage: LINT;
	{attribute 'FieldName' := 'acceleration_x'}
	acceleration_x: LINT;
	{attribute 'FieldName' := 'acceleration_y'}
	acceleration_y: LINT;
	{attribute 'FieldName' := 'acceleration_z'}
	acceleration_z: LINT;
	{attribute 'FieldName' := 'time_to_shutdown'}
	time_to_shutdown: LINT;
	{attribute 'FieldName' := 'fb_fw_rev'}
	fb_fw_rev: LINT;
END_STRUCT
END_TYPE

// ---- DUTs/ST_database_job_event.TcDUT
{attribute 'pack_mode' := '1'}
TYPE ST_database_job_event :
STRUCT
	datetime: ULINT;
	{attribute 'FieldName' := 'event_id'}
	event_id	: STRING;
	{attribute 'FieldName' := 'old_state'}
	old_state	: STRING;
	{attribute 'FieldName' := 'new_state'}
	new_state	: STRING;
	{attribute 'FieldName' := 'job_id'}
	{attribute 'TcEncoding':='UTF-8'}
	job_id		: STRING;
	{attribute 'TagName' := 'task_name'}
	{attribute 'TcEncoding':='UTF-8'}
	task_name	: STRING;
	{attribute 'FieldName' := 'error_id'}
	erro_id		: UDINT;
END_STRUCT
END_TYPE

// ---- DUTs/ST_mover_dynamics.TcDUT
{attribute 'pack_mode' := '1'}
TYPE ST_mover_dynamics :
STRUCT
	{attribute 'TagName' := 'title'}
	index: STRING;
	{attribute 'FieldName' := 'axis-a'}
	a: LREAL;
	{attribute 'FieldName' := 'axis-b'}
	b: LREAL;
	{attribute 'FieldName' := 'axis-c'}
	c: LREAL;
	{attribute 'FieldName' := 'axis-x'}
	x: LREAL;
	{attribute 'FieldName' := 'axis-y'}
	y: LREAL;
	{attribute 'FieldName' := 'axis-z'}
	z: LREAL;
END_STRUCT
END_TYPE

// ---- DUTs/ST_OperationPanel.TcDUT
TYPE ST_OperationPanel :
STRUCT
	bStart 						: BOOL;
	bEnable 					: BOOL;
	bDisable 					: BOOL;
	bReset 						: BOOL;
	bStop						: BOOL;
END_STRUCT
END_TYPE

// ---- DUTs/ST_RouterStatusInfo.TcDUT
{attribute 'pack_mode' := '1'}
TYPE ST_RouterStatusInfo :
STRUCT
	{attribute 'FieldName' := 'maxMem'}
	maxMem      : DWORD;(* Max. router memory byte size *)
	{attribute 'FieldName' := 'maxMemAvail'}
    maxMemAvail : DWORD;(* Available router memory byte size *)
	{attribute 'FieldName' := 'regPorts'}
    regPorts    : DWORD;(* Number of registered ports *)
	{attribute 'FieldName' := 'regDrivers'}
    regDrivers  : DWORD;(* Number of registered TwinCAT server ports *)
	{attribute 'FieldName' := 'amsDebugLog'}
    amsDebugLog : BOOL;(* TRUE = Ams logging/debugging enabled, FALSE = Ams logging/debugging disabled *)
END_STRUCT
END_TYPE

// ---- DUTs/TileInfoType.TcDUT
TYPE TileInfoType :
STRUCT
	Center 	: LREAL;
	East 	: LREAL;
	North 	: LREAL;
	South	: LREAL;
	West 	: LREAL;
	FanRPM	: UINT;
END_STRUCT
END_TYPE

// ---- GVLs/GVL.TcGVL
{attribute 'qualified_only'}
VAR_GLOBAL CONSTANT
	NUM_OF_MOVERS :UINT := 5;
	NUM_OF_TRACKS : UINT := 3;
	DB_MAX_COLUMNS : UDINT := 6;
	BUFFER_SIZE_DBWRITE : UINT := 500;
END_VAR
VAR_GLOBAL
	planar_movers	: ARRAY [1..NUM_OF_MOVERS] OF MC_PlanarMover;
	planar_environment : MC_PlanarEnvironment;
	planar_group	: MC_PlanarGroup;
	planar_tracks	: ARRAY [1..NUM_OF_TRACKS] OF MC_PlanarTrack;	
	// Database record driver
    //fbSQLRecorder 		:RecordSQL(DBID := 1);
    fbInfluxDBRecorder 		:RecordInfluxDB(DBID := 1);
	tf6420_enable	: BOOL;
END_VAR

// ---- POUs/MAIN.TcPOU
PROGRAM MAIN
VAR
	bStart 						: BOOL;
	bEnable 					: BOOL;
	bDisable 					: BOOL;
	bReset 						: BOOL;
	bStop						: BOOL;
	nCase 						: UINT;
	nDemoSequenceState			: UINT;
	
	cmdFB						: MC_PlanarFeedback;
	stMoverState				: MC_PLANAR_STATE;
	
	// Dynamic task creator
	fbMoveToPositionTaskCreator		: FB_TaskMoveToPosition_creator(GVL.planar_movers[1]);
	fbMoveCTaskCreator				: FB_TaskMoveC_creator(GVL.planar_movers[1]);
	fbMoveZTaskCreator				: FB_TaskMoveZ_creator(GVL.planar_movers[1]);
	fbMoveATaskCreator				: FB_TaskMoveA_tilt_creator(GVL.planar_movers[1]);
	fbMoveBTaskCreator				: FB_TaskMoveB_tilt_creator(GVL.planar_movers[1]);
	//batch_job_container_creator		: FB_BatchJobContainerCreator;
	fbJob							: jobmgmt.FB_Executor;
	
	random_gen : DRAND;
	random		:REAL;
	
	i: UINT;
	current_action : T_Maxstring;
	manual_command: iManualCommand;
	//ads_reporter : FB_ADSLOG_reporter;
	ads_reporter : FB_JobReporter;
	
	//試運転用パラメーター      
	(*          			
	Vel							: UDINT	:= 100;
	Acc							: UDINT	:= 1000;
	Dcc							: UDINT	:= 1000;
	Jerk						: UDINT	:= 5000;
	Ang_Vel						: UDINT	:= 100;
	Ang_Acc						: UDINT	:= 1000;
	Ang_Dcc						: UDINT	:= 1000;
	Ang_Jerk					: UDINT	:= 5000;
	*)             			
	 //デモ用パラメーター               			
	              			
	Vel							: UDINT	:= 400;
	Acc							: UDINT	:= 4000;
	Dcc							: UDINT	:= 4000;
	Jerk						: UDINT	:= 20000;
	Ang_Vel						: UDINT	:= 360;
	Ang_Acc						: UDINT	:= 3600;
	Ang_Dcc						: UDINT	:= 3600;
	Ang_Jerk					: UDINT	:= 36000;
	              			
	                			
	Height						: LREAL	:= 2.0;
	Cnt							: UINT;
	Z_High						: LREAL := 6.0;
	Z_Low						: LREAL := 2.0;
	A_Tilt						: LREAL := 0.0;
	B_Tilt						: LREAL := 0.0;
	Tilt						: LREAL := 2.5;
	Rotaion_Ang					: LREAL := 1.5;
	Estop						: BOOL;
	StopStep					: INT;
	fbDnyMoveEstop				: DynamicConstraint_PathXY;
	RotaionBit					: BOOL;
	Init_Angle					: BOOL;
	Init_Height_Tilt			: BOOL;
	
	Height_Tilt_Recover_Step	: INT;
	Init_Angle_Step				: INT;
	
	//  Utility Initial  -----------------------------------
	fbENviroment				: FB_TcIoXPlanarEnvironment;
	fbVisuXpalnar				: FB_XPlanarUtilityVisu;
	ipXpu						: I_TcIoXPlanarProcessingUnit;
	                			
	fbTcIoMover					: FB_TcIoXPlanarMover;
	ipXpm						: I_TcIoXPlanarMover;
	ipXpmsa						: I_XPlanarMoverScopeAdr;
	                			
	nStateInitXpu				: INT;
	bInit						: BOOL := FALSE;
	bInit_database				: BOOL := FALSE;

	LampTimer					: TON;
	ServoON						: BOOL;
	Error						: BOOL;
	Init_Start					: BOOL;

	
	Manupilate_Start: BOOL;
	nManupilationState: UINT;
	nJobConfigState: INT;
	Demo_Start: BOOL;
	manu_mode: BOOL;
	manual_command_event: BOOL;
	manual_command_event_mem: BOOL;
	manupilator_buttons: ARRAY [0..49] OF BOOL;
	manual_executor : REFERENCE TO FB_Executor;
	head : BOOL; tail: BOOL; order_num: UINT;
	Recipe_Display				: ARRAY [1..jobmgmt.ParamFuturesLib.MAX_TASK_NUM] OF T_MaxString;
	manual_start : BOOL;
	machine_mode: UINT;

	(* TF6420 Database server *)
    fbDtUtil : FB_DatetimeUtilities;

    // Record data buffer
    fb_database_job_event    :ST_database_job_event;    // 書込みデータ設定用
    database_job_event_buffer  :ARRAY [0..DbLibParam.DATA_BUFFER_SIZE - 1] OF ST_database_job_event; // バッファ配列の定義

    fb_job_event_db_recorder  :BufferedRecord(
        GVL.fbInfluxDBRecorder, 
        ADR(database_job_event_buffer)
    );		// record controller

	
	fb_home_job: INT;
	start: INT;
END_VAR
VAR PERSISTENT
	serial_num : UDINT;
END_VAR
VAR CONSTANT
	INIT_STEP	:	INT	 	:= 0;
	INIT_TILT 	: 	LREAL 	:= 0.0;
	INIT_HEIGHT :	LREAL 	:= 3.0;
	
END_VAR

//初期動作
IF NOT bInit THEN
		CASE nStateInitXpu OF
			0://Utilityの有効化
				IF fbENviroment.Init(TRUE) THEN
					fbENviroment.Init(FALSE);
					nStateInitXpu:=1;
				END_IF
			1://Utilityの実行を確認
				ipXpu:=fbENviroment.XpuTcIo(1);
				
				IF ipXpu<>0 THEN
					nStateInitXpu:=2;
				END_IF
				
			2://Job生成
				fbJob.continuous_mode := FALSE;
				fbJob.create_container(ContainerType.QUEUE, 'MAIN JOB');
				bInit := TRUE;
		END_CASE
	RETURN;
END_IF

IF NOT bInit_database THEN
	fb_job_event_db_recorder.min_chunk_size := 1;
	fb_job_event_db_recorder.max_chunk_size := 1;
	ads_reporter.fbDatabaseRecorder REF= fb_job_event_db_recorder;

	// Database column parameter initialization
	// 構造体名称の設定
	fb_job_event_db_recorder.set_buffer_info(
			struct_size := SIZEOF(database_job_event_buffer[0]), 
			buffer_size := SIZEOF(database_job_event_buffer), 
			structure_name := 'ST_database_job_event'); // Measurement name

	// SQLデータベースのテーブル名
	fb_job_event_db_recorder.SQL_parameters.table_name := 'job_event';

(*	
	// 列パラメータの登録
	fb_job_event_db_recorder.SQL_parameters.add_column(
		'datetime', 
		tf6420.E_ExpParameterType.Int64, 
		SIZEOF(fb_database_job_event.datetime)
	); // 列1
	fb_job_event_db_recorder.SQL_parameters.add_column(
		'old_state', 
		tf6420.E_ExpParameterType.STRING_,
		SIZEOF(fb_database_job_event.old_state)
	); // 列2
	fb_job_event_db_recorder.SQL_parameters.add_column(
		'new_status', 
		tf6420.E_ExpParameterType.STRING_,
		SIZEOF(fb_database_job_event.new_state)
	); // 列3
	fb_job_event_db_recorder.SQL_parameters.add_column(
		'task_name', 
		tf6420.E_ExpParameterType.STRING_, 
		SIZEOF(fb_database_job_event.task_name)
	); // 列4
	fb_job_event_db_recorder.SQL_parameters.add_column(
		'job_id', 
		tf6420.E_ExpParameterType.Int64, 
		SIZEOF(fb_database_job_event.job_id)
	); // 列5
	fb_job_event_db_recorder.SQL_parameters.add_column(
		'error_id', 
		tf6420.E_ExpParameterType.Int64, 
		SIZEOF(fb_database_job_event.erro_id)
	); // 列6
*)
	
	bInit_database := TRUE;
END_IF

GVL.planar_movers[1].Update();
cmdFB.Update();
ACT_Lamp_Ctrl();
stMoverState 					:= GVL.planar_movers[1].MCTOPLC.STD.State;

// SQL database
fbjob.job_event_reporter := ads_reporter;

//サーボオン
IF bEnable THEN
	GVL.planar_movers[1].Enable(cmdFB);
	bEnable := FALSE;
END_IF

//サーボオフ
IF bDisable THEN
	GVL.planar_movers[1].Disable(cmdFB);
	nDemoSequenceState := 0;
	nManupilationState := 0;
	nCase := 0;
	IF fbjob.reset() THEN
		bDisable	:= FALSE;
	END_IF
END_IF

//サーボオン＋動作ステップが０番の時にデモ動作開始
IF stMoverState = MC_PLANAR_STATE.Enabled THEN
	IF Init_Start AND nCase = 0 THEN
		// 原点復帰ボタンが押されたときの処理
		nCase 		:= 1;
		nManupilationState := 0;
		nDemoSequenceState := 0;
		Init_Start	:= FALSE;
	END_IF
	CASE nManupilationState OF
		0: // 待機状態
			IF manu_mode AND nDemoSequenceState = 0 AND nCase = 5 THEN
				// Manual Modeボタンが押された時の処理
				nCase := 0;
				nManupilationState := 1;
			ELSE
				manu_mode := FALSE;
			END_IF
			// avoid
		1: // Initialize jobs
			fbjob.create_container(ContainerType.QUEUE, 'MANUAL JOB');
			fbMoveToPositionTaskCreator.set_dynamics(Vel, Acc, Dcc, Jerk);
			fbMoveCTaskCreator.set_dynamics(Coord_Mcs_C1,Ang_Vel,Ang_Acc,Ang_Dcc,Ang_Jerk);
			fbMoveZTaskCreator.set_dynamics(Vel, Acc, Dcc, Jerk);
			fbMoveATaskCreator.set_dynamics(Vel, Acc, Dcc, Jerk);
			fbMoveBTaskCreator.set_dynamics(Vel, Acc, Dcc, Jerk);
			nManupilationState := 2;
		2:// 非同期タスク発行
			manual_command_event := FALSE;
			FOR i := 0 TO 49 DO
				// HMIボタン入力
				IF manupilator_buttons[i] THEN
					manual_command_event := TRUE; // イベントフラグ
					manual_command.i_com := i; // コマンド番号をMenualCommand型のenumへ変換（UNION）
				END_IF
			END_FOR
		
			IF manual_command_event AND NOT manual_command_event_mem THEN
				// イベントフラグ立ち上がり条件の作成
				CASE manual_command.com OF
					// コマンド番号毎にタスクをキューに登録
					ManualCommand.move_pos_c1:
						fbMoveToPositionTaskCreator.set_target_position(x := 240, y :=80, c :=0);
						fbjob.children.create_future(fbMoveToPositionTaskCreator,'MOVE C1');
					ManualCommand.move_pos_c2:
						fbMoveToPositionTaskCreator.set_target_position(x := 240, y :=120, c :=0);
						fbjob.children.create_future(fbMoveToPositionTaskCreator,'MOVE C2');
					ManualCommand.move_pos_c3:
						fbMoveToPositionTaskCreator.set_target_position(x := 240, y :=160, c :=0);
						fbjob.children.create_future(fbMoveToPositionTaskCreator,'MOVE C3');
					ManualCommand.move_pos_L1:
						fbMoveToPositionTaskCreator.set_target_position(x := 80, y :=80, c :=0);
						fbjob.children.create_future(fbMoveToPositionTaskCreator,'MOVE L1');
					ManualCommand.move_pos_L2:
						fbMoveToPositionTaskCreator.set_target_position(x := 80, y :=120, c :=0);
						fbjob.children.create_future(fbMoveToPositionTaskCreator,'MOVE L2');
					ManualCommand.move_pos_L3:
						fbMoveToPositionTaskCreator.set_target_position(x := 80, y :=160, c :=0);
						fbjob.children.create_future(fbMoveToPositionTaskCreator,'MOVE L3');
					ManualCommand.move_pos_r1:
						fbMoveToPositionTaskCreator.set_target_position(x := 400, y :=160, c :=0);
						fbjob.children.create_future(fbMoveToPositionTaskCreator,'MOVE R1');
					ManualCommand.move_pos_r2:
						fbMoveToPositionTaskCreator.set_target_position(x := 400, y :=120, c :=0);
						fbjob.children.create_future(fbMoveToPositionTaskCreator,'MOVE R2');
					ManualCommand.move_pos_r3:
						fbMoveToPositionTaskCreator.set_target_position(x := 400, y :=80, c :=0);
						fbjob.children.create_future(fbMoveToPositionTaskCreator,'MOVE R3');
					ManualCommand.move_roll_w:
						fbMoveCTaskCreator.set_target_position(270.0);
						fbjob.children.create_future(fbMoveCTaskCreator,'ROLL WEST');
					ManualCommand.move_roll_n:
						fbMoveCTaskCreator.set_target_position(0.0);
						fbjob.children.create_future(fbMoveCTaskCreator,'ROLL NORTH');
					ManualCommand.move_roll_e:
						fbMoveCTaskCreator.set_target_position(90.0);
						fbjob.children.create_future(fbMoveCTaskCreator,'ROLL EAST');
					ManualCommand.move_roll_s:
						fbMoveCTaskCreator.set_target_position(180.0);
						fbjob.children.create_future(fbMoveCTaskCreator,'ROLL SOUTH');
					ManualCommand.move_tilt_up_front:
						//fb_manu_job.add_future(fbMoveZTasks[1]);
						//fb_manu_job.add_future(fbMoveATasks[1]);					
					ManualCommand.move_tilt_up_rear:
						//fb_manu_job.add_future(fbMoveZTasks[1]);
						//fb_manu_job.add_future(fbMoveATasks[2]);					
					ManualCommand.move_tilt_up_right:
						//fb_manu_job.add_future(fbMoveZTasks[1]);
						//fb_manu_job.add_future(fbMoveBTasks[1]);
					ManualCommand.move_tilt_up_left:
						//fb_manu_job.add_future(fbMoveZTasks[1]);
						//fb_manu_job.add_future(fbMoveBTasks[2]);					
					ManualCommand.move_tilt_horizontal:
						//fb_manu_job.add_future(fbMoveATasks[3]);
						//fb_manu_job.add_future(fbMoveBTasks[3]);
						//fb_manu_job.add_future(fbMoveZTasks[2]);
					ManualCommand.move_up:
						//fb_manu_job.add_future(fbMoveZTasks[1]);
					ManualCommand.move_down:					
						//fb_manu_job.add_future(fbMoveZTasks[2]);
				END_CASE
			END_IF
			manual_command_event_mem := manual_command_event;

			//実行
			IF fbJob.ready THEN
				fbJob.start();
			END_IF
			IF fbJob.execute() AND fbJob.nErrorID = 0 THEN
				fbJob.init();
			END_IF
			//停止動作
			IF bStop THEN
				fbJob.abort();
			END_IF
			
			IF bReset THEN
				fbJob.start();
			END_IF
			//current_action := fbJob.active_future_id;
			
			IF fbJob.current_state = jobmgmt.E_FutureExecutionState.finish THEN
				nManupilationState := 2;				
			END_IF
			
			IF NOT manu_mode THEN
				nManupilationState := 1;
			END_IF
	END_CASE
END_IF


//原点復帰
CASE nCase OF
	0:
		// avoid step
		
	1: // job create
		CreateHomeJob(fbJob);
		IF fbJob.init() THEN
			nCase := 2;			
		END_IF
	2: // execute initialization
		IF fbJob.done AND fbJob.nErrorID = 0 THEN
			IF fbJob.init() THEN
				nCase := 5;			
			END_IF
		END_IF
	5: // Ready to start
		IF stMoverState = MC_PLANAR_STATE.Disabled THEN
			nCase := 0;
			nDemoSequenceState := 0;
		END_IF
END_CASE


//デモ動作開始
IF Demo_Start THEN
	IF nCase = 5 AND nDemoSequenceState = 0 THEN
		nDemoSequenceState 		:= 1;
	END_IF
END_IF


// デモ動作
CASE nDemoSequenceState OF
	0:
		// avoid
	1:
		IF serial_num = 16#FFFFFFFF THEN
			serial_num := 1;
		ELSE
			serial_num := serial_num + 1;
		END_IF
		
		
		CreateDemoJob_1(fbJob);
		nDemoSequenceState := 2;
	2:
		
		
		IF fbJob.done THEN
			IF fbJob.init() THEN
				IF Demo_Start THEN
					nDemoSequenceState := 1;
				ELSE
					nDemoSequenceState := 0;
				END_IF
			END_IF
		END_IF
		
END_CASE

IF nCase > 1 THEN
	//デモモード実行
	IF fbJob.ready THEN
		fbJob.start();
	END_IF
	//停止動作
	IF bStop THEN
		fbJob.abort();	
	END_IF
	IF fbJob.execute() THEN
		nCase := 0;
		nDemoSequenceState := 0;
	END_IF
END_IF


IF nDemoSequenceState > 0 THEN
	machine_mode := 6;
ELSIF nManupilationState > 0 THEN
	machine_mode := 7;
ELSIF nCase <= 5 THEN
	machine_mode := nCase;	
END_IF

IF bStop THEN
	bStop		:= FALSE;
END_IF


//動作とエラーリセット
IF bReset THEN
	GVL.planar_movers[1].Reset(cmdFB);
	IF fbJob.error_reset() THEN
		IF fbJob.resume() THEN
			bReset := FALSE;
		END_IF
	END_IF
END_IF

IoT();

ACTION ACT_Lamp_Ctrl:
Error := FALSE;

IF stMoverState = MC_PLANAR_STATE.Disabled THEN
	LampTimer.IN := NOT LampTimer.Q;
	LampTimer.PT := T#750MS;
	LampTimer();
	
	IF LampTimer.Q THEN
		ServoON := NOT ServoON;
		
	END_IF
ELSIF stMoverState = MC_PLANAR_STATE.Enabled THEN	
	ServoON := TRUE;

	
ELSIF stMoverState = MC_PLANAR_STATE.Error THEN	
	Error := TRUE;

END_IF
END_ACTION

METHOD CreateDemoJob_1 : BOOL
VAR_INPUT
	executor : REFERENCE TO FB_Executor;
END_VAR
VAR
	demo_job_container : InterfaceContainer;
	executor_item : REFERENCE TO FB_Executor;
	child_container : InterfaceContainer;
	i :UDINT;
END_VAR
demo_job_container := executor.children.create_container(ContainerType.BATCH, 'Demo Job').children;

fbMoveToPositionTaskCreator.set_dynamics(Vel, Acc, Dcc, Jerk);
fbMoveCTaskCreator.set_dynamics(Coord_Mcs_C1,Ang_Vel,Ang_Acc,Ang_Dcc,Ang_Jerk);
fbMoveZTaskCreator.set_dynamics(Vel, Acc, Dcc, Jerk);
fbMoveATaskCreator.set_dynamics(Vel, Acc, Dcc, Jerk);
fbMoveBTaskCreator.set_dynamics(Vel, Acc, Dcc, Jerk);

executor_item REF= demo_job_container.create_container(ContainerType.BATCH, '<POSITIONING>');
executor_item.init();
child_container := executor_item.children;

fbMoveToPositionTaskCreator.set_target_position(x := 240, y :=120, c :=0);
child_container.create_future(fbMoveToPositionTaskCreator, 'Move B2');
fbMoveToPositionTaskCreator.set_target_position(x := 80, y :=80, c :=0);
child_container.create_future(fbMoveToPositionTaskCreator, 'Move A3');
fbMoveToPositionTaskCreator.set_target_position(x := 80, y :=160, c :=0);
child_container.create_future(fbMoveToPositionTaskCreator, 'Move A1');
fbMoveToPositionTaskCreator.set_target_position(x := 400, y :=160, c :=0);
child_container.create_future(fbMoveToPositionTaskCreator, 'Move C1');
fbMoveToPositionTaskCreator.set_target_position(x := 400, y :=80, c :=0);
child_container.create_future(fbMoveToPositionTaskCreator, 'Move C3');
fbMoveToPositionTaskCreator.set_target_position(x := 240, y :=120, c :=0);
child_container.create_future(fbMoveToPositionTaskCreator, 'Move B2');

executor_item REF= demo_job_container.create_container(ContainerType.BATCH,  '<ROTATING>');
executor_item.init();
child_container := executor_item.children;

fbMoveCTaskCreator.set_target_position(360.0);
child_container.create_future(fbMoveCTaskCreator, 'ROLL 360.0 deg');
fbMoveCTaskCreator.set_target_position(0.0);
child_container.create_future(fbMoveCTaskCreator, 'ROLL 0.0 deg');

executor_item REF= demo_job_container.create_container(ContainerType.BATCH,  '<ELEVATION>');
executor_item.init();
child_container := executor_item.children;

FOR i := 1 TO 9 DO
	fbMoveZTaskCreator.set_target_position(Z_High);
	child_container.create_future(fbMoveZTaskCreator, 'ELEV. UP');
	fbMoveZTaskCreator.set_target_position(Z_Low);
	child_container.create_future(fbMoveZTaskCreator, 'ELEV. DOWN');
END_FOR


executor_item REF= demo_job_container.create_container(ContainerType.BATCH,  '<TILT F/B>');
executor_item.init();
child_container := executor_item.children;

fbMoveZTaskCreator.set_target_position(Z_High);
child_container.create_future(fbMoveZTaskCreator, 'ELEV. UP');

FOR i := 1 TO 10 DO
	fbMoveATaskCreator.set_target_position(Tilt);
	child_container.create_future(fbMoveATaskCreator, 'Tilt forwards');
	fbMoveATaskCreator.set_target_position(-Tilt);
	child_container.create_future(fbMoveATaskCreator, 'Tilt backwards');
END_FOR
fbMoveATaskCreator.set_target_position(0);
child_container.create_future(fbMoveATaskCreator, 'F/B tilt holizontal');

executor_item REF= demo_job_container.create_container(ContainerType.BATCH, '<TILT L/R>');
executor_item.init();
child_container := executor_item.children;

fbMoveZTaskCreator.set_target_position(Z_High);
child_container.create_future(fbMoveZTaskCreator, 'ELEV. UP');

FOR i := 1 TO 10 DO
	fbMoveBTaskCreator.set_target_position(Tilt);
	child_container.create_future(fbMoveBTaskCreator, 'Tilt forwards');
	fbMoveBTaskCreator.set_target_position(-Tilt);
	child_container.create_future(fbMoveBTaskCreator, 'Tilt backwards');
END_FOR
fbMoveBTaskCreator.set_target_position(0);
child_container.create_future(fbMoveBTaskCreator, 'L/R tilt holizontal');



executor_item REF= demo_job_container.create_container(ContainerType.BATCH, '<TILT L/R>');
executor_item.init();
child_container := executor_item.children;

fbMoveZTaskCreator.set_target_position(Z_High);
child_container.create_future(fbMoveZTaskCreator, 'ELEV. UP');

FOR i := 1 TO 4 DO
	fbMoveATaskCreator.set_target_position(Rotaion_Ang);
	child_container.create_future(fbMoveATaskCreator, 'Tilt forwards');
	fbMoveBTaskCreator.set_target_position(Rotaion_Ang);
	child_container.create_future(fbMoveBTaskCreator, 'Tilt forwards');
	fbMoveATaskCreator.set_target_position(-Rotaion_Ang);
	child_container.create_future(fbMoveATaskCreator, 'Tilt backwards');
	fbMoveBTaskCreator.set_target_position(-Rotaion_Ang);
	child_container.create_future(fbMoveBTaskCreator, 'Tilt backwards');
END_FOR
fbMoveATaskCreator.set_target_position(0);
child_container.create_future(fbMoveATaskCreator, 'F/B tilt holizontal');
fbMoveBTaskCreator.set_target_position(0);
child_container.create_future(fbMoveBTaskCreator, 'L/R tilt holizontal');
fbMoveZTaskCreator.set_target_position(INIT_HEIGHT);
child_container.create_future(fbMoveZTaskCreator, 'Height initial position.');
END_METHOD

METHOD CreateDemoJob_2 : BOOL
VAR_INPUT
	container : InterfaceContainer;
END_VAR
VAR
	demo_job_container: jobmgmt.InterfaceContainer;
	executor_item : REFERENCE TO FB_Executor;
	child_container : InterfaceContainer;
	i :UDINT;
END_VAR
executor_item REF= container.create_container(ContainerType.BATCH, 'Demo Job');
demo_job_container := executor_item.children;

fbMoveToPositionTaskCreator.set_dynamics(Vel, Acc, Dcc, Jerk);
fbMoveCTaskCreator.set_dynamics(Coord_Mcs_C1,Ang_Vel,Ang_Acc,Ang_Dcc,Ang_Jerk);
fbMoveZTaskCreator.set_dynamics(Vel, Acc, Dcc, Jerk);
fbMoveATaskCreator.set_dynamics(Vel, Acc, Dcc, Jerk);
fbMoveBTaskCreator.set_dynamics(Vel, Acc, Dcc, Jerk);

executor_item REF= demo_job_container.create_future(jobmgmt.GVL.batch_job_container_creator, '<POSITIONING>');
executor_item.init();
child_container := executor_item.children;

fbMoveToPositionTaskCreator.set_target_position(x := 240, y :=120, c :=0);
child_container.create_future(fbMoveToPositionTaskCreator, 'Move B2');
fbMoveToPositionTaskCreator.set_target_position(x := 80, y :=80, c :=0);
child_container.create_future(fbMoveToPositionTaskCreator, 'Move A3');
fbMoveToPositionTaskCreator.set_target_position(x := 80, y :=160, c :=0);
child_container.create_future(fbMoveToPositionTaskCreator, 'Move A1');
fbMoveToPositionTaskCreator.set_target_position(x := 400, y :=160, c :=0);
child_container.create_future(fbMoveToPositionTaskCreator, 'Move C1');
fbMoveToPositionTaskCreator.set_target_position(x := 400, y :=80, c :=0);
child_container.create_future(fbMoveToPositionTaskCreator, 'Move C3');
fbMoveToPositionTaskCreator.set_target_position(x := 240, y :=120, c :=0);
child_container.create_future(fbMoveToPositionTaskCreator, 'Move B2');
fbMoveToPositionTaskCreator.set_target_position(x := 240, y :=120, c :=0);
child_container.create_future(fbMoveToPositionTaskCreator, 'Move B2');
fbMoveToPositionTaskCreator.set_target_position(x := 80, y :=80, c :=0);
child_container.create_future(fbMoveToPositionTaskCreator, 'Move A3');
fbMoveToPositionTaskCreator.set_target_position(x := 80, y :=160, c :=0);
child_container.create_future(fbMoveToPositionTaskCreator, 'Move A1');
fbMoveToPositionTaskCreator.set_target_position(x := 400, y :=160, c :=0);
child_container.create_future(fbMoveToPositionTaskCreator, 'Move C1');
fbMoveToPositionTaskCreator.set_target_position(x := 400, y :=80, c :=0);
child_container.create_future(fbMoveToPositionTaskCreator, 'Move C3');
fbMoveToPositionTaskCreator.set_target_position(x := 240, y :=120, c :=0);
child_container.create_future(fbMoveToPositionTaskCreator, 'Move B2');

executor_item REF= demo_job_container.create_future(jobmgmt.GVL.batch_job_container_creator, '<ROTATING>');
executor_item.init();
child_container := executor_item.children;

FOR i := 5 TO 360 BY 5 DO
	fbMoveCTaskCreator.set_target_position(UDINT_TO_LREAL(i));
	child_container.create_future(fbMoveCTaskCreator, CONCAT('ROLL' , TO_STRING(i)));	
END_FOR
fbMoveCTaskCreator.set_target_position(0);
child_container.create_future(fbMoveCTaskCreator, 'ROLL 0 deg');

executor_item REF= demo_job_container.create_future(jobmgmt.GVL.batch_job_container_creator, '<ELEVATION>');
executor_item.init();
child_container := executor_item.children;

FOR i := 1 TO 9 DO
	fbMoveZTaskCreator.set_target_position(Z_High);
	child_container.create_future(fbMoveZTaskCreator, 'ELEV. UP');
	fbMoveZTaskCreator.set_target_position(Z_Low);
	child_container.create_future(fbMoveZTaskCreator, 'ELEV. DOWN');
END_FOR


executor_item REF= demo_job_container.create_future(jobmgmt.GVL.batch_job_container_creator, '<TILT F/B>');
executor_item.init();
child_container := executor_item.children;

fbMoveZTaskCreator.set_target_position(Z_High);
child_container.create_future(fbMoveZTaskCreator, 'ELEV. UP');

FOR i := 1 TO 10 DO
	fbMoveATaskCreator.set_target_position(Tilt);
	child_container.create_future(fbMoveATaskCreator, 'Tilt forwards');
	fbMoveATaskCreator.set_target_position(-Tilt);
	child_container.create_future(fbMoveATaskCreator, 'Tilt backwards');
END_FOR
fbMoveATaskCreator.set_target_position(0);
child_container.create_future(fbMoveATaskCreator, 'F/B tilt holizontal');

executor_item REF= demo_job_container.create_future(jobmgmt.GVL.batch_job_container_creator, '<TILT L/R>');
executor_item.init();
child_container := executor_item.children;

fbMoveZTaskCreator.set_target_position(Z_High);
child_container.create_future(fbMoveZTaskCreator, 'ELEV. UP');

FOR i := 1 TO 10 DO
	fbMoveBTaskCreator.set_target_position(Tilt);
	child_container.create_future(fbMoveBTaskCreator, 'Tilt forwards');
	fbMoveBTaskCreator.set_target_position(-Tilt);
	child_container.create_future(fbMoveBTaskCreator, 'Tilt backwards');
END_FOR
fbMoveBTaskCreator.set_target_position(0);
child_container.create_future(fbMoveBTaskCreator, 'L/R tilt holizontal');



executor_item REF= demo_job_container.create_future(jobmgmt.GVL.batch_job_container_creator, '<TILT L/R>');
executor_item.init();
child_container := executor_item.children;

fbMoveZTaskCreator.set_target_position(Z_High);
child_container.create_future(fbMoveZTaskCreator, 'ELEV. UP');

FOR i := 1 TO 4 DO
	fbMoveATaskCreator.set_target_position(Rotaion_Ang);
	child_container.create_future(fbMoveATaskCreator, 'Tilt forwards');
	fbMoveBTaskCreator.set_target_position(Rotaion_Ang);
	child_container.create_future(fbMoveBTaskCreator, 'Tilt forwards');
	fbMoveATaskCreator.set_target_position(-Rotaion_Ang);
	child_container.create_future(fbMoveATaskCreator, 'Tilt backwards');
	fbMoveBTaskCreator.set_target_position(-Rotaion_Ang);
	child_container.create_future(fbMoveBTaskCreator, 'Tilt backwards');
END_FOR
fbMoveATaskCreator.set_target_position(0);
child_container.create_future(fbMoveATaskCreator, 'F/B tilt holizontal');
fbMoveBTaskCreator.set_target_position(0);
child_container.create_future(fbMoveBTaskCreator, 'L/R tilt holizontal');
fbMoveZTaskCreator.set_target_position(INIT_HEIGHT);
child_container.create_future(fbMoveZTaskCreator, 'Height initial position.');
END_METHOD

METHOD CreateDemoJob_3 : BOOL
VAR_INPUT
	container : InterfaceContainer;
END_VAR
VAR
	demo_job_container: jobmgmt.InterfaceContainer;
	executor_item : REFERENCE TO FB_Executor;
	child_container : InterfaceContainer;
	i :UDINT;
END_VAR
executor_item REF= container.create_container(ContainerType.BATCH, 'Demo Job');
demo_job_container := executor_item.children;

fbMoveToPositionTaskCreator.set_dynamics(Vel, Acc, Dcc, Jerk);
fbMoveCTaskCreator.set_dynamics(Coord_Mcs_C1,Ang_Vel,Ang_Acc,Ang_Dcc,Ang_Jerk);
fbMoveZTaskCreator.set_dynamics(Vel, Acc, Dcc, Jerk);
fbMoveATaskCreator.set_dynamics(Vel, Acc, Dcc, Jerk);
fbMoveBTaskCreator.set_dynamics(Vel, Acc, Dcc, Jerk);

executor_item REF= demo_job_container.create_future(jobmgmt.GVL.batch_job_container_creator, '<POSITIONING>');
executor_item.init();
child_container := executor_item.children;

fbMoveToPositionTaskCreator.set_target_position(x := 240, y :=120, c :=0);
child_container.create_future(fbMoveToPositionTaskCreator, 'Move B2');
fbMoveToPositionTaskCreator.set_target_position(x := 80, y :=80, c :=0);
child_container.create_future(fbMoveToPositionTaskCreator, 'Move A3');
fbMoveToPositionTaskCreator.set_target_position(x := 80, y :=160, c :=0);
child_container.create_future(fbMoveToPositionTaskCreator, 'Move A1');
fbMoveToPositionTaskCreator.set_target_position(x := 400, y :=160, c :=0);
child_container.create_future(fbMoveToPositionTaskCreator, 'Move C1');
fbMoveToPositionTaskCreator.set_target_position(x := 400, y :=80, c :=0);
child_container.create_future(fbMoveToPositionTaskCreator, 'Move C3');
fbMoveToPositionTaskCreator.set_target_position(x := 240, y :=120, c :=0);
child_container.create_future(fbMoveToPositionTaskCreator, 'Move B2');

executor_item REF= demo_job_container.create_future(jobmgmt.GVL.batch_job_container_creator, '<ROTATING>');
executor_item.init();
child_container := executor_item.children;

fbMoveCTaskCreator.set_target_position(360.0);
child_container.create_future(fbMoveCTaskCreator, 'ROLL 360.0 deg');
fbMoveCTaskCreator.set_target_position(0.0);
child_container.create_future(fbMoveCTaskCreator, 'ROLL 0.0 deg');

executor_item REF= demo_job_container.create_future(jobmgmt.GVL.batch_job_container_creator, '<ELEVATION>');
executor_item.init();
child_container := executor_item.children;

FOR i := 1 TO 9 DO
	fbMoveZTaskCreator.set_target_position(Z_High);
	child_container.create_future(fbMoveZTaskCreator, 'ELEV. UP');
	fbMoveZTaskCreator.set_target_position(Z_Low);
	child_container.create_future(fbMoveZTaskCreator, 'ELEV. DOWN');
END_FOR


executor_item REF= demo_job_container.create_future(jobmgmt.GVL.batch_job_container_creator, '<TILT F/B>');
executor_item.init();
child_container := executor_item.children;

fbMoveZTaskCreator.set_target_position(Z_High);
child_container.create_future(fbMoveZTaskCreator, 'ELEV. UP');

FOR i := 1 TO 10 DO
	fbMoveATaskCreator.set_target_position(Tilt);
	child_container.create_future(fbMoveATaskCreator, 'Tilt forwards');
	fbMoveATaskCreator.set_target_position(-Tilt);
	child_container.create_future(fbMoveATaskCreator, 'Tilt backwards');
END_FOR
fbMoveATaskCreator.set_target_position(0);
child_container.create_future(fbMoveATaskCreator, 'F/B tilt holizontal');

executor_item REF= demo_job_container.create_future(jobmgmt.GVL.batch_job_container_creator, '<TILT L/R>');
executor_item.init();
child_container := executor_item.children;

fbMoveZTaskCreator.set_target_position(Z_High);
child_container.create_future(fbMoveZTaskCreator, 'ELEV. UP');

FOR i := 1 TO 10 DO
	fbMoveBTaskCreator.set_target_position(Tilt);
	child_container.create_future(fbMoveBTaskCreator, 'Tilt forwards');
	fbMoveBTaskCreator.set_target_position(-Tilt);
	child_container.create_future(fbMoveBTaskCreator, 'Tilt backwards');
END_FOR
fbMoveBTaskCreator.set_target_position(0);
child_container.create_future(fbMoveBTaskCreator, 'L/R tilt holizontal');



executor_item REF= demo_job_container.create_future(jobmgmt.GVL.batch_job_container_creator, '<TILT L/R>');
executor_item.init();
child_container := executor_item.children;

fbMoveZTaskCreator.set_target_position(Z_High);
child_container.create_future(fbMoveZTaskCreator, 'ELEV. UP');

FOR i := 1 TO 4 DO
	fbMoveATaskCreator.set_target_position(Rotaion_Ang);
	child_container.create_future(fbMoveATaskCreator, 'Tilt forwards');
	fbMoveBTaskCreator.set_target_position(Rotaion_Ang);
	child_container.create_future(fbMoveBTaskCreator, 'Tilt forwards');
	fbMoveATaskCreator.set_target_position(-Rotaion_Ang);
	child_container.create_future(fbMoveATaskCreator, 'Tilt backwards');
	fbMoveBTaskCreator.set_target_position(-Rotaion_Ang);
	child_container.create_future(fbMoveBTaskCreator, 'Tilt backwards');
END_FOR
fbMoveATaskCreator.set_target_position(0);
child_container.create_future(fbMoveATaskCreator, 'F/B tilt holizontal');
fbMoveBTaskCreator.set_target_position(0);
child_container.create_future(fbMoveBTaskCreator, 'L/R tilt holizontal');
fbMoveZTaskCreator.set_target_position(INIT_HEIGHT);
child_container.create_future(fbMoveZTaskCreator, 'Height initial position.');
END_METHOD

METHOD CreateHomeJob : BOOL
VAR_INPUT
	executor : REFERENCE TO FB_Executor;
END_VAR
VAR
	home_job_container: jobmgmt.InterfaceContainer;
	executor_item : REFERENCE TO FB_Executor;
	child_container : InterfaceContainer;
	i :UDINT;
END_VAR
home_job_container := executor.children.create_container(ContainerType.BATCH, 'Home Job').children;

fbMoveToPositionTaskCreator.set_dynamics(Vel, Acc, Dcc, Jerk);
fbMoveCTaskCreator.set_dynamics(Coord_Mcs_C1,Ang_Vel,Ang_Acc,Ang_Dcc,Ang_Jerk);
fbMoveZTaskCreator.set_dynamics(Vel, Acc, Dcc, Jerk);
fbMoveATaskCreator.set_dynamics(Vel, Acc, Dcc, Jerk);
fbMoveBTaskCreator.set_dynamics(Vel, Acc, Dcc, Jerk);

fbMoveBTaskCreator.set_target_position(0);
home_job_container.create_future(fbMoveBTaskCreator, 'L/R tilt holizontal');

fbMoveATaskCreator.set_target_position(0);
home_job_container.create_future(fbMoveATaskCreator, 'F/B tilt holizontal');

fbMoveZTaskCreator.set_target_position(INIT_HEIGHT);
home_job_container.create_future(fbMoveZTaskCreator, 'Height initial position.');

fbMoveCTaskCreator.set_target_position(0.0);
home_job_container.create_future(fbMoveCTaskCreator, 'ROLL 0.0 deg');

fbMoveToPositionTaskCreator.set_dynamics(Vel, Acc, Dcc, Jerk);
fbMoveToPositionTaskCreator.set_target_position(x := 240, y :=120, c :=0);
home_job_container.create_future(fbMoveToPositionTaskCreator, 'Move center position');
END_METHOD

METHOD MakeTasks : InterfaceFuture
VAR_INPUT
END_VAR
VAR
		demo_job_container: InterfaceContainer;
END_VAR
(*
IF fbJob.reset() THEN
	fbJob.future := fbJob.create_future(FB_BatchJobContainerCreator, 'Demo Job');
	fbJob.init();
	demo_job_container := fbJob.children;
END_IF
fbMoveToPositionTaskCreator.set_dynamics(Vel, Acc, Dcc, Jerk);
fbMoveToPositionTaskCreator.set_target_position(x := 240, y :=120, c :=0);
demo_job_container.create_future(fbMoveToPositionTaskCreator, 'Move B2');
fbMoveToPositionTaskCreator.set_target_position(x := 80, y :=80, c :=0);
demo_job_container.create_future(fbMoveToPositionTaskCreator, 'Move A3');
fbMoveToPositionTaskCreator.set_target_position(x := 80, y :=160, c :=0);
demo_job_container.create_future(fbMoveToPositionTaskCreator, 'Move A1');
fbMoveToPositionTaskCreator.set_target_position(x := 400, y :=160, c :=0);
demo_job_container.create_future(fbMoveToPositionTaskCreator, 'Move C1');
fbMoveToPositionTaskCreator.set_target_position(x := 400, y :=80, c :=0);
demo_job_container.create_future(fbMoveToPositionTaskCreator, 'Move C3');
fbMoveToPositionTaskCreator.set_target_position(x := 80, y :=120, c :=0);
demo_job_container.create_future(fbMoveToPositionTaskCreator, 'Move A2');
fbMoveToPositionTaskCreator.set_target_position(x := 240, y :=80, c :=0);
demo_job_container.create_future(fbMoveToPositionTaskCreator, 'Move B3');
fbMoveToPositionTaskCreator.set_target_position(x := 240, y :=160, c :=0);
demo_job_container.create_future(fbMoveToPositionTaskCreator, 'Move B1');
fbMoveToPositionTaskCreator.set_target_position(x := 240, y :=160, c :=0);
demo_job_container.create_future(fbMoveToPositionTaskCreator, 'Move B1');
fbMoveToPositionTaskCreator.set_target_position(x := 400, y :=120, c :=0);
demo_job_container.create_future(fbMoveToPositionTaskCreator, 'Move C2');


// 回転動作タスク追加
fbMoveCTaskCreator.set_dynamics(Coord_Mcs_C1,Ang_Vel,Ang_Acc,Ang_Dcc,Ang_Jerk);
fbMoveCTaskCreator.set_target_position(0.0);
demo_job_container.create_future(fbMoveCTaskCreator, 'ROLL 0.0 deg');
fbMoveCTaskCreator.set_target_position(360.0);
demo_job_container.create_future(fbMoveCTaskCreator, 'ROLL 360.0 deg');
fbMoveCTaskCreator.set_target_position(90.0);
demo_job_container.create_future(fbMoveCTaskCreator, 'ROLL 90.0 deg');
fbMoveCTaskCreator.set_target_position(180.0);
demo_job_container.create_future(fbMoveCTaskCreator, 'ROLL 180.0 deg');
fbMoveCTaskCreator.set_target_position(270.0);
demo_job_container.create_future(fbMoveCTaskCreator, 'ROLL 27.0 deg');



// 上下動作タスク追加
fbMoveZTaskCreator.set_dynamics(Vel, Acc, Dcc, Jerk);
fbMoveZTaskCreator.set_target_position(Z_High);
demo_job_container.create_future(fbMoveZTaskCreator, 'ELEV. UP');
fbMoveZTaskCreator.set_target_position(Z_Low);
demo_job_container.create_future(fbMoveZTaskCreator, 'ELEV. DOWN');
fbMoveZTaskCreator.set_target_position(INIT_HEIGHT);
demo_job_container.create_future(fbMoveZTaskCreator, 'Height initial position.');

// 傾きA動作タスク追加
fbMoveATaskCreator.set_dynamics(Vel, Acc, Dcc, Jerk);
fbMoveATaskCreator.set_target_position(Tilt);
demo_job_container.create_future(fbMoveATaskCreator, 'Tilt forwards');
fbMoveATaskCreator.set_target_position(-Tilt);
demo_job_container.create_future(fbMoveATaskCreator, 'Tilt backwards');
fbMoveATaskCreator.set_target_position(0);
demo_job_container.create_future(fbMoveATaskCreator, 'F/B tilt holizontal');


// 傾きB動作タスク追加
fbMoveBTaskCreator.set_dynamics(Vel, Acc, Dcc, Jerk);
fbMoveBTaskCreator.set_target_position(Tilt);
demo_job_container.create_future(fbMoveBTaskCreator, 'Tilt right');
fbMoveBTaskCreator.set_target_position(-Tilt);
demo_job_container.create_future(fbMoveBTaskCreator, 'Tilt left');
fbMoveBTaskCreator.set_target_position(0);
demo_job_container.create_future(fbMoveBTaskCreator, 'L/R tilt horizontal');
*)
END_METHOD

END_PROGRAM

// ---- POUs/model/activities/FB_TaskMoveToPosition_creator.TcPOU
FUNCTION_BLOCK FB_TaskMoveToPosition_creator IMPLEMENTS InterfaceTaskCreator
VAR_INPUT
END_VAR
VAR_OUTPUT
END_VAR
VAR
	_x				: MC_LREAL;
	_y				: MC_LREAL;
	_c				: MC_LREAL;
	_v				: MC_LREAL;
	_a				: MC_LREAL;
	_d				: MC_LREAL;
	_j				: MC_LREAL;
	_mover			: REFERENCE TO MC_PlanarMover;
END_VAR

{warning 'add method implementation '}
METHOD create_future : jobmgmt.InterfaceFuture
VAR_INPUT
	future_name	: STRING;
END_VAR
VAR
	_p_future : POINTER TO FB_TaskMoveToPosition;
END_VAR
_p_future := __NEW(FB_TaskMoveToPosition);
_p_future^.mover REF= _mover;
_p_future^.future_name := future_name;
_p_future^.set_dynamics(_v,_a,_d,_j);
_p_future^.set_target_position(_x, _y, _c);
create_future := _p_future^;
END_METHOD

{warning 'add method implementation '}
METHOD destroy_future : InterfaceFuture
VAR_INPUT
	future	: jobmgmt.InterfaceFuture;
END_VAR
VAR
	_p_future : POINTER TO FB_TaskMoveToPosition;
END_VAR
IF __QUERYPOINTER(future, _p_future) THEN
	__DELETE(_p_future);
	IF _p_future = 0  THEN
		destroy_future := 0;
	END_IF
END_IF
END_METHOD

METHOD FB_init : BOOL
VAR_INPUT
	bInitRetains : BOOL; // if TRUE, the retain variables are initialized (warm start / cold start)
	bInCopyCode : BOOL;  // if TRUE, the instance afterwards gets moved into the copy code (online change)
	mover : REFERENCE TO MC_PlanarMover;
END_VAR
_mover REF= mover;
END_METHOD

METHOD set_dynamics : BOOL
VAR_INPUT
	v: MC_LREAL;
	a: MC_LREAL;
	d: MC_LREAL;
	j: MC_LREAL;
END_VAR
_v := v;
_a := a;
_d := d;
_j := j;
set_dynamics := TRUE;
END_METHOD

METHOD set_target_position : BOOL
VAR_INPUT
	x: LREAL;
	y: LREAL;
	c: LREAL;
END_VAR
_x := x;
_y := y;
_c := c;

set_target_position := TRUE;
END_METHOD

END_FUNCTION_BLOCK

// ---- POUs/model/activities/FB_TaskMoveToPosition.TcPOU
{attribute 'enable_dynamic_creation'}
FUNCTION_BLOCK FB_TaskMoveToPosition EXTENDS FB_AbstructFuture
VAR_OUTPUT
END_VAR
VAR
	_v				: MC_LREAL;
	_a				: MC_LREAL;
	_d				: MC_LREAL;
	_j				: MC_LREAL;
	_pos_x 			: LREAL;
	_pos_y 			: LREAL;
	_pos_c			: LREAL;
	_dynamics		: DynamicConstraint_PathXY;
	_position 		: PositionXYC;
	_error_id		: UDINT;
	_mover		: REFERENCE TO MC_PlanarMover;
	_cmdFB			: MC_PlanarFeedback;
	_prohibit 		: BOOL;
	_abort_executor : FB_Executor;
	_state_num 			:UINT;
	_abort_state	:UINT;
END_VAR

{warning 'add method implementation '}
METHOD abort : BOOL
_cmdFB.Update();
_state_num := 0;
CASE _abort_state OF
	0:
		IF _cmdFB.Active THEN
			_dynamics.SetValuesVADJ(2000,20000,200000,200000);
			_abort_state := 1;
		ELSE
			abort := TRUE;
		END_IF
	1:
		//停止
		_mover.Halt(_cmdFB,_dynamics);
		_abort_state := 2;
	2:
		//停止完了フラグ待ち
		IF _cmdFB.Done THEN
			abort := TRUE;
			_error_id := 0;
		END_IF
		IF _cmdFB.Error THEN
			abort := TRUE;
			_error_id := _cmdFB.ErrorId;
		END_IF
END_CASE
END_METHOD

{warning 'add method implementation '}
METHOD execute : BOOL
_cmdFB.Update();
_abort_state := 0;
CASE _state_num OF
	0:
		//直線運動
		IF NOT _cmdFB.Active AND NOT _cmdFB.Busy THEN
			_mover.MoveToPosition(_cmdFB,_position,_dynamics,0);
			_state_num := 1;
		END_IF
	1:
		//直線運動の完了フラグ待ち
		IF _cmdFB.Done THEN
			execute := TRUE;
			_error_id := 0;
		END_IF
		IF _cmdFB.Error THEN
			execute := TRUE;
			_error_id := _cmdFB.ErrorId;
		END_IF
END_CASE
END_METHOD

{warning 'add method implementation '}
METHOD init : BOOL
IF _prohibit THEN
	_error_id := 16#80000000;
	init := TRUE;
ELSIF _v = 0 OR _a = 0 OR _d = 0 THEN
	_error_id := 1;
	init := TRUE;
ELSE
	_dynamics.SetValuesVADJ(_v, _a, _d, _j);
	_position.SetValuesXYC(_pos_x, _pos_y, _pos_c);
	_abort_executor.init();
	_error_id := 0;
	_state_num := 0;
	_abort_state := 0;
	init := TRUE;
END_IF
END_METHOD

PROPERTY mover : REFERENCE TO MC_PlanarMover
SET
_mover REF= mover;
END_SET
END_PROPERTY

{warning 'add property implementation'}
PROPERTY nErrorID : UDINT
GET
nErrorID := _error_id;
END_GET
END_PROPERTY

{warning 'add method implementation '}
METHOD quit : BOOL
init();
quit := TRUE;
END_METHOD

METHOD set_dynamics : BOOL
VAR_INPUT
	v: MC_LREAL;
	a: MC_LREAL;
	d: MC_LREAL;
	j: MC_LREAL;
END_VAR
_v := v;
_a := a;
_d := d;
_j := j;
set_dynamics := TRUE;
END_METHOD

METHOD set_target_position : BOOL
VAR_INPUT
	x: LREAL;
	y: LREAL;
	c: LREAL;
END_VAR
_pos_x := x;
_pos_y := y;
_pos_c := c;

set_target_position := TRUE;
END_METHOD

END_FUNCTION_BLOCK

// ---- POUs/model/activities/FB_TaskMoveC_creator.TcPOU
FUNCTION_BLOCK FB_TaskMoveC_creator IMPLEMENTS InterfaceTaskCreator
VAR_INPUT
END_VAR
VAR_OUTPUT
END_VAR
VAR
	_coordinate		: CoordinateType;
	_p				: MC_LREAL;
	_v				: MC_LREAL;
	_a				: MC_LREAL;
	_d				: MC_LREAL;
	_j				: MC_LREAL;
	_dynamics		: DynamicConstraint_Coordinates;
	_coptions		: ST_MoveCOptions;
	_additional_turns: UDINT;
	_direction: MC_DIRECTION;
	_mover			: REFERENCE TO MC_PlanarMover;
END_VAR

{warning 'add method implementation '}
METHOD create_future : jobmgmt.InterfaceFuture
VAR_INPUT
	future_name	: STRING;
END_VAR
VAR
	_p_future : POINTER TO FB_TaskMoveC;
END_VAR
_p_future := __NEW(FB_TaskMoveC);
_p_future^.mover REF= _mover;
_p_future^.future_name := future_name;
_p_future^.set_options(_additional_turns,_direction);
_p_future^.set_dynamics(_coordinate,_v,_a,_d,_j);
_p_future^.set_target_position(_p);
create_future := _p_future^;
END_METHOD

{warning 'add method implementation '}
METHOD destroy_future : InterfaceFuture
VAR_INPUT
	future	: jobmgmt.InterfaceFuture;
END_VAR
VAR
	_p_future : POINTER TO FB_TaskMoveC;
END_VAR
IF __QUERYPOINTER(future, _p_future) THEN
	__DELETE(_p_future);
	IF _p_future = 0  THEN
		destroy_future := 0;
	END_IF
END_IF
END_METHOD

METHOD FB_init : BOOL
VAR_INPUT
	bInitRetains : BOOL; // if TRUE, the retain variables are initialized (warm start / cold start)
	bInCopyCode : BOOL;  // if TRUE, the instance afterwards gets moved into the copy code (online change)
	mover : REFERENCE TO MC_PlanarMover;
END_VAR
_mover REF= mover;
END_METHOD

METHOD set_dynamics : BOOL
VAR_INPUT
	coordinate: CoordinateType;
	v: MC_LREAL;
	a: MC_LREAL;
	d: MC_LREAL;
	j: MC_LREAL;
END_VAR
_coordinate := coordinate;
_v := v;
_a := a;
_d := d;
_j := j;
set_dynamics := TRUE;
END_METHOD

METHOD set_options : BOOL
VAR_INPUT
	(* Addition turns to move in modulo movement (positive or negative). *)
	additional_turns : UDINT := 0;
	(* Direction in which the target is approached. *)
	 {attribute 'GUID' := 'FA9CA56B-5BDF-42DB-BC74-B14868EB8B42'}
	direction : MC_DIRECTION := MC_DIRECTION.mcDirectionNonModulo;
END_VAR
_coptions.additionalTurns := additional_turns;
_coptions.direction := direction;
set_options := TRUE;
END_METHOD

METHOD set_target_position : BOOL
VAR_INPUT
	c: LREAL;
END_VAR
_p := c;
set_target_position := TRUE;
END_METHOD

END_FUNCTION_BLOCK

// ---- POUs/model/activities/FB_TaskMoveC.TcPOU
{attribute 'enable_dynamic_creation'}
FUNCTION_BLOCK FB_TaskMoveC EXTENDS FB_AbstructFuture
VAR_OUTPUT
END_VAR
VAR
	_coordinate		: CoordinateType;
	_v				: MC_LREAL;
	_a				: MC_LREAL;
	_d				: MC_LREAL;
	_j				: MC_LREAL;
	_dynamics		: DynamicConstraint_Coordinates;
	_coptions		: ST_MoveCOptions;
	_position 		: LREAL;
	_error_id		: UDINT;
	_mover			: REFERENCE TO MC_PlanarMover;
	_cmdFB			: MC_PlanarFeedback;
	_prohibit 		: BOOL;
	_abort_executor : FB_Executor;
	_state_num 			:UINT;
	_abort_state	:UINT;
END_VAR

{warning 'add method implementation '}
METHOD abort : BOOL
_cmdFB.Update();
_state_num := 0;
CASE _abort_state OF
	0:
		IF _cmdFB.Active THEN
			_dynamics.SetLimit(_coordinate,2000,20000,200000,200000);
			_abort_state := 1;
		ELSE
			abort := TRUE;
		END_IF
	1:
		//停止
		_mover.Halt(_cmdFB,_dynamics);
		_abort_state := 2;
	2:
		//停止完了フラグ待ち
		IF _cmdFB.Done THEN
			abort := TRUE;
			_error_id := 0;
		END_IF
		IF _cmdFB.Error THEN
			abort := TRUE;
			_error_id := _cmdFB.ErrorId;
		END_IF
END_CASE
END_METHOD

{warning 'add method implementation '}
METHOD execute : BOOL
_cmdFB.Update();
_abort_state := 0;
CASE _state_num OF
	0:
		//直線運動
		IF NOT _cmdFB.Active AND NOT _cmdFB.Busy THEN
			_mover.MoveC(_cmdFB,_position,_dynamics,_coptions);
			_state_num := 1;
		END_IF
	1:
		//直線運動の完了フラグ待ち
		IF _cmdFB.Done THEN
			execute := TRUE;
			_error_id := 0;
		END_IF
		IF _cmdFB.Error THEN
			execute := TRUE;
			_error_id := _cmdFB.ErrorId;
		END_IF
END_CASE
END_METHOD

{warning 'add method implementation '}
METHOD init : BOOL
IF _prohibit THEN
	_error_id := 16#80000000;
	init := TRUE;
ELSIF _v = 0 OR _a = 0 OR _d = 0 THEN
	_error_id := 1;
	init := TRUE;
ELSE
	_dynamics.SetLimit(_coordinate, _v, _a, _d, _j);
	_abort_executor.init();
	_error_id := 0;
	_state_num := 0;
	_abort_state := 0;
	init := TRUE;
END_IF
END_METHOD

PROPERTY mover : REFERENCE TO MC_PlanarMover
SET
_mover REF= mover;
END_SET
END_PROPERTY

{warning 'add property implementation'}
PROPERTY nErrorID : UDINT
GET
nErrorID := _error_id;
END_GET
END_PROPERTY

{warning 'add method implementation '}
METHOD quit : BOOL
init();
quit := TRUE;
END_METHOD

METHOD set_dynamics : BOOL
VAR_INPUT
	coordinate: CoordinateType;
	v: MC_LREAL;
	a: MC_LREAL;
	d: MC_LREAL;
	j: MC_LREAL;
END_VAR
_coordinate := coordinate;
_v := v;
_a := a;
_d := d;
_j := j;
set_dynamics := TRUE;
END_METHOD

METHOD set_options : BOOL
VAR_INPUT
	(* Addition turns to move in modulo movement (positive or negative). *)
	additional_turns : UDINT := 0;
	(* Direction in which the target is approached. *)
	 {attribute 'GUID' := 'FA9CA56B-5BDF-42DB-BC74-B14868EB8B42'}
	direction : MC_DIRECTION := MC_DIRECTION.mcDirectionNonModulo;
END_VAR
_coptions.additionalTurns := additional_turns;
_coptions.direction := direction;
set_options := TRUE;
END_METHOD

METHOD set_target_position : BOOL
VAR_INPUT
	c: LREAL;
END_VAR
_position := c;
set_target_position := TRUE;
END_METHOD

END_FUNCTION_BLOCK

// ---- POUs/model/activities/FB_TaskMoveZ_creator.TcPOU
FUNCTION_BLOCK FB_TaskMoveZ_creator IMPLEMENTS InterfaceTaskCreator
VAR_INPUT
END_VAR
VAR_OUTPUT
END_VAR
VAR
	_p				: MC_LREAL;
	_v				: MC_LREAL;
	_a				: MC_LREAL;
	_d				: MC_LREAL;
	_j				: MC_LREAL;
	_mover			: REFERENCE TO MC_PlanarMover;
END_VAR

{warning 'add method implementation '}
METHOD create_future : jobmgmt.InterfaceFuture
VAR_INPUT
	future_name	: STRING;
END_VAR
VAR
	_p_future : POINTER TO FB_TaskMoveZ;
END_VAR
_p_future := __NEW(FB_TaskMoveZ);
_p_future^.mover REF= _mover;
_p_future^.future_name := future_name;
_p_future^.set_dynamics(_v,_a,_d,_j);
_p_future^.set_target_position(_p);
create_future := _p_future^;
END_METHOD

{warning 'add method implementation '}
METHOD destroy_future : InterfaceFuture
VAR_INPUT
	future	: jobmgmt.InterfaceFuture;
END_VAR
VAR
	_p_future : POINTER TO FB_TaskMoveZ;
END_VAR
IF __QUERYPOINTER(future, _p_future) THEN
	__DELETE(_p_future);
	IF _p_future = 0  THEN
		destroy_future := 0;
	END_IF
END_IF
END_METHOD

METHOD FB_init : BOOL
VAR_INPUT
	bInitRetains : BOOL; // if TRUE, the retain variables are initialized (warm start / cold start)
	bInCopyCode : BOOL;  // if TRUE, the instance afterwards gets moved into the copy code (online change)
	mover : REFERENCE TO MC_PlanarMover;
END_VAR
_mover REF= mover;
END_METHOD

METHOD set_dynamics : BOOL
VAR_INPUT
	v: MC_LREAL;
	a: MC_LREAL;
	d: MC_LREAL;
	j: MC_LREAL;
END_VAR
_v := v;
_a := a;
_d := d;
_j := j;
set_dynamics := TRUE;
END_METHOD

METHOD set_target_position : BOOL
VAR_INPUT
	z: LREAL;
END_VAR
_p := z;

set_target_position := TRUE;
END_METHOD

END_FUNCTION_BLOCK

// ---- POUs/model/activities/FB_TaskMoveZ.TcPOU
{attribute 'enable_dynamic_creation'}
FUNCTION_BLOCK FB_TaskMoveZ EXTENDS FB_AbstructFuture
VAR_OUTPUT
END_VAR
VAR
	_v				: MC_LREAL;
	_a				: MC_LREAL;
	_d				: MC_LREAL;
	_j				: MC_LREAL;
	_dynamics		: DynamicConstraint_PathXY;
	_position 		: LREAL;
	_error_id		: UDINT;
	_mover			: REFERENCE TO MC_PlanarMover;
	_cmdFB			: MC_PlanarFeedback;
	_prohibit 		: BOOL;
	_abort_executor : FB_Executor;
	_state_num 			:UINT;
	_abort_state	:UINT;
END_VAR

{warning 'add method implementation '}
METHOD abort : BOOL
_cmdFB.Update();
_state_num := 0;
CASE _abort_state OF
	0:
		IF _cmdFB.Active THEN
			_dynamics.SetValuesVADJ(2000,20000,200000,200000);
			_abort_state := 1;
		ELSE
			abort := TRUE;
		END_IF
	1:
		//停止
		_mover.Halt(_cmdFB,_dynamics);
		_abort_state := 2;
	2:
		//停止完了フラグ待ち
		IF _cmdFB.Done THEN
			abort := TRUE;
			_error_id := 0;
		END_IF
		IF _cmdFB.Error THEN
			abort := TRUE;
			_error_id := _cmdFB.ErrorId;
		END_IF
END_CASE
END_METHOD

{warning 'add method implementation '}
METHOD execute : BOOL
_cmdFB.Update();
_abort_state := 0;
CASE _state_num OF
	0:
		//直線運動
		IF NOT _cmdFB.Active AND NOT _cmdFB.Busy THEN
			_mover.MoveZ(_cmdFB,_position,_dynamics);
			_state_num := 1;
		END_IF
	1:
		//直線運動の完了フラグ待ち
		IF _cmdFB.Done THEN
			execute := TRUE;
			_error_id := 0;
		END_IF
		IF _cmdFB.Error THEN
			execute := TRUE;
			_error_id := _cmdFB.ErrorId;
		END_IF
END_CASE
END_METHOD

{warning 'add method implementation '}
METHOD init : BOOL
IF _prohibit THEN
	_error_id := 16#80000000;
	init := TRUE;
ELSIF _v = 0 OR _a = 0 OR _d = 0 THEN
	_error_id := 1;
	init := TRUE;
ELSE
	_dynamics.SetValuesVADJ(_v, _a, _d, _j);
	_abort_executor.init();
	_error_id := 0;
	_state_num := 0;
	_abort_state := 0;
	init := TRUE;
END_IF
END_METHOD

PROPERTY mover : REFERENCE TO MC_PlanarMover
SET
_mover REF= mover;
END_SET
END_PROPERTY

{warning 'add property implementation'}
PROPERTY nErrorID : UDINT
GET
nErrorID := _error_id;
END_GET
END_PROPERTY

{warning 'add method implementation '}
METHOD quit : BOOL
init();
quit := TRUE;
END_METHOD

METHOD set_dynamics : BOOL
VAR_INPUT
	v: MC_LREAL;
	a: MC_LREAL;
	d: MC_LREAL;
	j: MC_LREAL;
END_VAR
_v := v;
_a := a;
_d := d;
_j := j;
set_dynamics := TRUE;
END_METHOD

METHOD set_target_position : BOOL
VAR_INPUT
	z: LREAL;
END_VAR
_position := z;

set_target_position := TRUE;
END_METHOD

END_FUNCTION_BLOCK

// ---- POUs/model/activities/FB_TaskMoveA_tilt_Creator.TcPOU
FUNCTION_BLOCK FB_TaskMoveA_tilt_Creator IMPLEMENTS InterfaceTaskCreator
VAR_INPUT
END_VAR
VAR_OUTPUT
END_VAR
VAR
	_p				: MC_LREAL;
	_v				: MC_LREAL;
	_a				: MC_LREAL;
	_d				: MC_LREAL;
	_j				: MC_LREAL;
	_mover			: REFERENCE TO MC_PlanarMover;
END_VAR

{warning 'add method implementation '}
METHOD create_future : jobmgmt.InterfaceFuture
VAR_INPUT
	future_name	: STRING;
END_VAR
VAR
	_p_future : POINTER TO FB_TaskMoveA_tilt;
END_VAR
_p_future := __NEW(FB_TaskMoveA_tilt);
_p_future^.mover REF= _mover;
_p_future^.future_name := future_name;
_p_future^.set_dynamics(_v,_a,_d,_j);
_p_future^.set_target_position(_p);
create_future := _p_future^;
END_METHOD

{warning 'add method implementation '}
METHOD destroy_future : InterfaceFuture
VAR_INPUT
	future	: jobmgmt.InterfaceFuture;
END_VAR
VAR
	_p_future : POINTER TO FB_TaskMoveA_tilt;
END_VAR
IF __QUERYPOINTER(future, _p_future) THEN
	__DELETE(_p_future);
	IF _p_future = 0  THEN
		destroy_future := 0;
	END_IF
END_IF
END_METHOD

METHOD FB_init : BOOL
VAR_INPUT
	bInitRetains : BOOL; // if TRUE, the retain variables are initialized (warm start / cold start)
	bInCopyCode : BOOL;  // if TRUE, the instance afterwards gets moved into the copy code (online change)
	mover : REFERENCE TO MC_PlanarMover;
END_VAR
_mover REF= mover;
END_METHOD

METHOD set_dynamics : BOOL
VAR_INPUT
	v: MC_LREAL;
	a: MC_LREAL;
	d: MC_LREAL;
	j: MC_LREAL;
END_VAR
_v := v;
_a := a;
_d := d;
_j := j;
set_dynamics := TRUE;
END_METHOD

METHOD set_target_position : BOOL
VAR_INPUT
	position: LREAL;
END_VAR
_p := position;
END_METHOD

END_FUNCTION_BLOCK

// ---- POUs/model/activities/FB_TaskMoveA_tilt.TcPOU
{attribute 'enable_dynamic_creation'}
FUNCTION_BLOCK FB_TaskMoveA_tilt EXTENDS FB_AbstructFuture
VAR_OUTPUT
END_VAR
VAR
	_v				: MC_LREAL;
	_a				: MC_LREAL;
	_d				: MC_LREAL;
	_j				: MC_LREAL;
	_dynamics		: DynamicConstraint_PathXY;
	_position 		: LREAL;
	_error_id		: UDINT;
	_mover			: REFERENCE TO MC_PlanarMover;
	_cmdFB			: MC_PlanarFeedback;
	_prohibit 		: BOOL;
	_abort_executor : FB_Executor;
	_state_num 			:UINT;
	_abort_state	:UINT;
END_VAR

{warning 'add method implementation '}
METHOD abort : BOOL
VAR_INST
	home_a :BOOL;
	home_b :BOOL;
END_VAR
_cmdFB.Update();
_state_num :=0;
CASE _abort_state OF
	0:
		IF _cmdFB.Active THEN
			_dynamics.SetValuesVADJ(2000,20000,200000,200000);
			home_a := FALSE;
			home_b := FALSE;
			//停止
			_mover.Halt(_cmdFB,_dynamics);
			_abort_state := 1;
		ELSE
			abort := TRUE;
		END_IF
	1:
		IF _cmdFB.Done THEN
			IF _cmdFB.Error THEN
				abort := TRUE;
				_abort_state := 0;
				_error_id := _cmdFB.ErrorId;
			ELSE
				IF NOT home_a THEN
					_abort_state := 2;
				ELSIF NOT home_b THEN
					_abort_state := 3;
				ELSE
					abort := TRUE;
					_error_id := 0;
				END_IF
			END_IF
		END_IF
	2:
		_mover.MoveA(_cmdFB,0,_dynamics);
		home_a := TRUE;
		_abort_state := 1;
	3:
		_mover.MoveB(_cmdFB,0,_dynamics);
		home_b := TRUE;
		_abort_state := 1;
END_CASE
END_METHOD

{warning 'add method implementation '}
METHOD execute : BOOL
_cmdFB.Update();
_abort_state := 0;
CASE _state_num OF
	0:
		//直線運動
		IF NOT _cmdFB.Active AND NOT _cmdFB.Busy THEN
			_mover.MoveA(_cmdFB,_position,_dynamics);
			_state_num := 1;
		END_IF
	1:
		//直線運動の完了フラグ待ち
		IF _cmdFB.Done THEN
			execute := TRUE;
			_error_id := 0;
		END_IF
		IF _cmdFB.Error THEN
			execute := TRUE;
			_error_id := _cmdFB.ErrorId;
		END_IF
END_CASE
END_METHOD

{warning 'add method implementation '}
METHOD init : BOOL
IF _prohibit THEN
	_error_id := 16#80000000;
	init := TRUE;
ELSIF _v = 0 OR _a = 0 OR _d = 0 THEN
	_error_id := 1;
	init := TRUE;
ELSE
	_dynamics.SetValuesVADJ(_v, _a, _d, _j);
	_abort_executor.init();
	_error_id := 0;
	_state_num := 0;
	_abort_state := 0;
	init := TRUE;
END_IF
END_METHOD

PROPERTY mover : REFERENCE TO MC_PlanarMover
SET
_mover REF= mover;
END_SET
END_PROPERTY

{warning 'add property implementation'}
PROPERTY nErrorID : UDINT
GET
nErrorID := _error_id;
END_GET
END_PROPERTY

{warning 'add method implementation '}
METHOD quit : BOOL
init();
quit := TRUE;
END_METHOD

METHOD set_dynamics : BOOL
VAR_INPUT
	v: MC_LREAL;
	a: MC_LREAL;
	d: MC_LREAL;
	j: MC_LREAL;
END_VAR
_v := v;
_a := a;
_d := d;
_j := j;
set_dynamics := TRUE;
END_METHOD

METHOD set_target_position : BOOL
VAR_INPUT
	z: LREAL;
END_VAR
_position := z;
set_target_position := TRUE;
END_METHOD

END_FUNCTION_BLOCK

// ---- POUs/model/activities/FB_TaskMoveB_tilt_creator.TcPOU
FUNCTION_BLOCK FB_TaskMoveB_tilt_creator IMPLEMENTS InterfaceTaskCreator
VAR_INPUT
END_VAR
VAR_OUTPUT
END_VAR
VAR
	_p				: MC_LREAL;
	_v				: MC_LREAL;
	_a				: MC_LREAL;
	_d				: MC_LREAL;
	_j				: MC_LREAL;
	_mover			: REFERENCE TO MC_PlanarMover;
END_VAR

{warning 'add method implementation '}
METHOD create_future : jobmgmt.InterfaceFuture
VAR_INPUT
	future_name	: STRING;
END_VAR
VAR
	_p_future : POINTER TO FB_TaskMoveB_tilt;
END_VAR
_p_future := __NEW(FB_TaskMoveB_tilt);
_p_future^.mover REF= _mover;
_p_future^.future_name := future_name;
_p_future^.set_dynamics(_v,_a,_d,_j);
_p_future^.set_target_position(_p);
create_future := _p_future^;
END_METHOD

{warning 'add method implementation '}
METHOD destroy_future : InterfaceFuture
VAR_INPUT
	future	: jobmgmt.InterfaceFuture;
END_VAR
VAR
	_p_future : POINTER TO FB_TaskMoveB_tilt;
END_VAR
IF __QUERYPOINTER(future, _p_future) THEN
	__DELETE(_p_future);
	IF _p_future = 0  THEN
		destroy_future := 0;
	END_IF
END_IF
END_METHOD

METHOD FB_init : BOOL
VAR_INPUT
	bInitRetains : BOOL; // if TRUE, the retain variables are initialized (warm start / cold start)
	bInCopyCode : BOOL;  // if TRUE, the instance afterwards gets moved into the copy code (online change)
	mover : REFERENCE TO MC_PlanarMover;
END_VAR
_mover REF= mover;
END_METHOD

METHOD set_dynamics : BOOL
VAR_INPUT
	v: MC_LREAL;
	a: MC_LREAL;
	d: MC_LREAL;
	j: MC_LREAL;
END_VAR
_v := v;
_a := a;
_d := d;
_j := j;
set_dynamics := TRUE;
END_METHOD

METHOD set_target_position : BOOL
VAR_INPUT
	z: LREAL;
END_VAR
_p := z;
set_target_position := TRUE;
END_METHOD

END_FUNCTION_BLOCK

// ---- POUs/model/activities/FB_TaskMoveB_tilt.TcPOU
{attribute 'enable_dynamic_creation'}
FUNCTION_BLOCK FB_TaskMoveB_tilt EXTENDS FB_AbstructFuture
VAR_OUTPUT
END_VAR
VAR
	_v				: MC_LREAL;
	_a				: MC_LREAL;
	_d				: MC_LREAL;
	_j				: MC_LREAL;
	_dynamics		: DynamicConstraint_PathXY;
	_position 		: LREAL;
	_error_id		: UDINT;
	_mover			: REFERENCE TO MC_PlanarMover;
	_cmdFB			: MC_PlanarFeedback;
	_prohibit 		: BOOL;
	_abort_executor : FB_Executor;
	_state_num 			:UINT;
	_abort_state	:UINT;
END_VAR

{warning 'add method implementation '}
METHOD abort : BOOL
VAR_INST
	home_a :BOOL;
	home_b :BOOL;
END_VAR
_cmdFB.Update();
_state_num :=0;
CASE _abort_state OF
	0:
		IF _cmdFB.Active THEN
			_dynamics.SetValuesVADJ(2000,20000,200000,200000);
			home_a := FALSE;
			home_b := FALSE;
			//停止
			_mover.Halt(_cmdFB,_dynamics);
			_abort_state := 1;
		ELSE
			abort := TRUE;
		END_IF
	1:
		IF _cmdFB.Done THEN
			IF _cmdFB.Error THEN
				abort := TRUE;
				_abort_state := 0;
				_error_id := _cmdFB.ErrorId;
			ELSE
				IF NOT home_a THEN
					_abort_state := 2;
				ELSIF NOT home_b THEN
					_abort_state := 3;
				ELSE
					abort := TRUE;
					_error_id := 0;
				END_IF
			END_IF
		END_IF
	2:
		_mover.MoveA(_cmdFB,0,_dynamics);
		home_a := TRUE;
		_abort_state := 1;
	3:
		_mover.MoveB(_cmdFB,0,_dynamics);
		home_b := TRUE;
		_abort_state := 1;
END_CASE
END_METHOD

{warning 'add method implementation '}
METHOD execute : BOOL
_cmdFB.Update();
_abort_state := 0;
CASE _state_num OF
	0:
		//直線運動
		IF NOT _cmdFB.Active AND NOT _cmdFB.Busy THEN
			_mover.MoveB(_cmdFB,_position,_dynamics);
			_state_num := 1;
		END_IF
	1:
		//直線運動の完了フラグ待ち
		IF _cmdFB.Done THEN
			execute := TRUE;
			_error_id := 0;
		END_IF
		IF _cmdFB.Error THEN
			execute := TRUE;
			_error_id := _cmdFB.ErrorId;
		END_IF
END_CASE
END_METHOD

METHOD init : BOOL
IF _prohibit THEN
	_error_id := 16#80000000;
	init := TRUE;
ELSIF _v = 0 OR _a = 0 OR _d = 0 THEN
	_error_id := 1;
	init := TRUE;
ELSE
	_dynamics.SetValuesVADJ(_v, _a, _d, _j);
	_abort_executor.init();
	_error_id := 0;
	_state_num := 0;
	_abort_state := 0;
	init := TRUE;
END_IF
END_METHOD

PROPERTY mover : REFERENCE TO MC_PlanarMover
SET
_mover REF= mover;
END_SET
END_PROPERTY

{warning 'add property implementation'}
PROPERTY nErrorID : UDINT
GET
nErrorID := _error_id;
END_GET
END_PROPERTY

{warning 'add method implementation '}
METHOD quit : BOOL
init();
quit := TRUE;
END_METHOD

METHOD set_dynamics : BOOL
VAR_INPUT
	v: MC_LREAL;
	a: MC_LREAL;
	d: MC_LREAL;
	j: MC_LREAL;
END_VAR
_v := v;
_a := a;
_d := d;
_j := j;
set_dynamics := TRUE;
END_METHOD

METHOD set_target_position : BOOL
VAR_INPUT
	z: LREAL;
END_VAR
_position := z;

set_target_position := TRUE;
END_METHOD

END_FUNCTION_BLOCK

// ---- POUs/model/IoT/FB_JobReporter.TcPOU
FUNCTION_BLOCK FB_JobReporter IMPLEMENTS InterfaceObserver
VAR_INPUT
END_VAR
VAR_OUTPUT
	event : JobEventReport;
	executing : JobEventReport;
	scope_task_triggers: ARRAY [0..10] OF BOOL;
	log_view: ARRAY [0..3, 0..19] OF T_MaxString;
	db_record_data : ST_database_job_event;
END_VAR
VAR
	_fbDatabaseRecorder : REFERENCE TO BufferedRecord;
END_VAR

METHOD _record_scope : BOOL
VAR_INPUT
	event : JobEventReport;
END_VAR

IF event.task_name = 'Tilt forwards' THEN
		IF event.new_state = 'process' THEN
			scope_task_triggers[0] := TRUE;
		ELSIF event.new_state = 'quit' THEN
			scope_task_triggers[0] := FALSE;
		END_IF
END_IF
END_METHOD

METHOD _record_sqldb : BOOL
VAR_INPUT
	event : JobEventReport;
END_VAR
END_METHOD

PROPERTY fbDatabaseRecorder : REFERENCE TO BufferedRecord
SET
_fbDatabaseRecorder REF= fbDatabaseRecorder;
END_SET
END_PROPERTY

{warning 'add method implementation '}
METHOD subscribe_job_directory : BOOL
VAR_INPUT
	executor	: REFERENCE TO jobmgmt.FB_Executor;
END_VAR

VAR
	job_log: T_MaxString;
END_VAR

job_log := CONCAT(job_log, 'JOB STRUCTURE');
IF executor.future <> 0 THEN
	job_log := CONCAT(job_log, '/ FUTURE_NAME : ');
	job_log := CONCAT(job_log, executor.future.future_name);
	job_log := CONCAT(job_log, ', ');	
END_IF
job_log := CONCAT(job_log, 'JOB_ID : ');
job_log := CONCAT(job_log, executor.id);

ADSLOGSTR(msgCtrlMask := ADSLOG_MSGTYPE_LOG, msgFmtStr := job_log, strArg := '');
END_METHOD

METHOD subscribe_job_event : BOOL
VAR_INPUT
	(* Subject text of event*)
	subject	: jobmgmt.T_MaxString;
	(* Job state before transition.*)
	old_state	: jobmgmt.E_FutureExecutionState;
	(* Job state after transition.*)
	new_state	: jobmgmt.E_FutureExecutionState;
	(* File-time at the time of transition.*)
	record_time	: jobmgmt.T_FILETIME64;
	(* Reference to job instance of which transition occurs.*)
	executor	: REFERENCE TO jobmgmt.FB_Executor;
END_VAR
VAR
	text : T_MaxString;
END_VAR
VAR_INST
	fb_timezone_info : FB_GetTimeZoneInformation := (bExecute := TRUE);
    // Datetime utilities
    fbDtUtil : FB_DatetimeUtilities;
END_VAR
//For log
event.old_state := TO_STRING(old_state);
event.new_state := TO_STRING(new_state);
event.record_time := FILETIME64_TO_ISO8601(fileTime := record_time, nBias := DINT_TO_INT(fb_timezone_info.tzInfo.bias), bUTC := TRUE,nPrecision := 6);
event.job_id := executor.id;
event.task_name := executor.future.future_name;
event.erro_id := executor.nErrorID;

// _record_scope(event);
//_record_sqldb(event);

IF new_state = E_FutureExecutionState.process THEN
	executing := event;
END_IF

IF old_state = E_FutureExecutionState.process OR new_state = E_FutureExecutionState.process THEN

	// Report to ADS Log
	text := event.record_time;
	text := CONCAT(text, '	');
	text := CONCAT(text, event.new_state);
	text := CONCAT(text, '		');
	text := CONCAT(text, event.task_name);
	text := CONCAT(text, '		');
	text := CONCAT(text, event.job_id);
	ADSLOGSTR(msgCtrlMask := ADSLOG_MSGTYPE_LOG, msgFmtStr := text, strArg := '');	

	
	// Report to HMI
	MEMCPY(ADR(log_view[0,1]), ADR(log_view[0,0]), SIZEOF(log_view[0,0]) * 19);
	MEMCPY(ADR(log_view[1,1]), ADR(log_view[1,0]), SIZEOF(log_view[0,0]) * 19);
	MEMCPY(ADR(log_view[2,1]), ADR(log_view[2,0]), SIZEOF(log_view[0,0]) * 19);
	MEMCPY(ADR(log_view[3,1]), ADR(log_view[3,0]), SIZEOF(log_view[0,0]) * 19);
	log_view[0,0] := event.record_time;
	log_view[1,0] := event.task_name;
	IF old_state = E_FutureExecutionState.process THEN
		log_view[2,0] := 'END';
	ELSE
		log_view[2,0] := 'START';
	END_IF
	log_view[3,0] := event.job_id;
	
END_IF


// For Database
// Windowsの時刻ロケールデータとの同期等を行うため常時実行
fbDtUtil();

IF __ISVALIDREF(_fbDatabaseRecorder) THEN
	// 記録用の構造体へのデータ登録
	// fbDtUtil.Filetime_To_UnixT()でマイクロ秒精度のUNIX時間を取得する
	db_record_data.datetime := fbDtUtil.Filetime_To_UnixT(F_GetSystemTime());
	db_record_data.event_id := subject;
	db_record_data.old_state := event.old_state;
	db_record_data.new_state := event.new_state;
	db_record_data.task_name := event.task_name;
	db_record_data.job_id := event.job_id;
	db_record_data.erro_id := executor.nErrorID;
	
	IF GVL.tf6420_enable THEN
		_fbDatabaseRecorder.write(ADR(db_record_data));			
	END_IF
END_IF

subscribe_job_event := TRUE;
END_METHOD

END_FUNCTION_BLOCK

// ---- POUs/IoT.TcPOU
PROGRAM IoT
VAR CONSTANT
	EC_MASTER_NETID : T_AmsNetId := '192.168.80.1.4.1';
END_VAR
VAR
	
	//TileInfo					: ARRAY [0..1] OF TileInfoType;

	sdo_controller : FB_CoeSdoAccess(sNetId := EC_MASTER_NETID);
	planar_tiles_diag_data : ARRAY[1..2] OF sdo_xplanar_aps_diag;
	sessions: ARRAY [1..2] OF CoeSdoCommand;
	read_cycle_timer: TON;
	fbMqttPublish : FB_mqtt_publish;
	
	slave_state : FB_EcGetSlaveState;
	state : ST_EcSlaveStateBits;
	
	// Diag data dabase recorder
	database_aps_diag_buffer  :ARRAY [0..1999] OF ST_database_aps_diag; // バッファ配列の定義
    fb_aps_diag_db_recorder  :BufferedRecord(
        GVL.fbInfluxDBRecorder, 
        ADR(database_aps_diag_buffer)
    );		// record controller

	// XPlanar dynamics data recorder
	database_mover_dynamics_buffer  :ARRAY [0..9999] OF ST_mover_dynamics; // バッファ配列の定義
    fb_mover_dynamics_recorder  :BufferedRecord(
        GVL.fbInfluxDBRecorder, 
        ADR(database_mover_dynamics_buffer)
    );		// record controller

	// ADS Router information tracing
	database_ads_router_info_buffer : ARRAY [0..499] OF ST_RouterStatusInfo;
	fb_ads_router_status_recorder : BufferedRecord(
		GVL.fbInfluxDBRecorder, 
		ADR(database_ads_router_info_buffer)
	);
	
	record_data_set_positions : ST_mover_dynamics := (index := 'Mover 1 Setting position');
	record_data_act_positions : ST_mover_dynamics := (index := 'Mover 1 Actual position');
	
	db_initialize :BOOL;
	structure_size: INT;
	SetDynamics : CDT_MCTOPLC_PLANAR_MOVER_SET;
	ActDynamics : CDT_MCTOPLC_PLANAR_MOVER_ACT;
	
	ads_router_status_record_interval_timer : TON := (PT:=T#1S);

	fb_get_router_status : FB_GetRouterStatusInfo;
	fb_get_router_status_report : BOOL;
	router_status_record_data : ST_RouterStatusInfo;
	
END_VAR

// Database Writing actions
GVL.fbInfluxDBRecorder();

//Xplanar各タイルの温度情報の取得
//FB_ECCoeSdoReadを使ったライブラリTwinCATDiagnosisToolsにてCoEアクセスするので、こちらはコメントアウト
(*
IF fbENviroment.XpuTcIo(1).TileCoE(1,1).DiagData.Update() THEN
	TileInfo[0].Center 	:= fbENviroment.XpuTcIo(1).TileCoE(1,1).DiagData.TemperatureCenter;
	TileInfo[0].East 	:= fbENviroment.XpuTcIo(1).TileCoE(1,1).DiagData.TemperatureEast;
	TileInfo[0].North 	:= fbENviroment.XpuTcIo(1).TileCoE(1,1).DiagData.TemperatureNorth;
	TileInfo[0].South 	:= fbENviroment.XpuTcIo(1).TileCoE(1,1).DiagData.TemperatureSouth;
	TileInfo[0].West 	:= fbENviroment.XpuTcIo(1).TileCoE(1,1).DiagData.TemperatureWest;
	TileInfo[0].FanRPM	:= fbENviroment.XpuTcIo(1).TileCoE(1,1).DiagData.FanRpm;
	
END_IF;

IF fbENviroment.XpuTcIo(1).TileCoE(1,2).DiagData.Update() THEN
	TileInfo[1].Center 	:= fbENviroment.XpuTcIo(1).TileCoE(1,2).DiagData.TemperatureCenter;
	TileInfo[1].East 	:= fbENviroment.XpuTcIo(1).TileCoE(1,2).DiagData.TemperatureEast;
	TileInfo[1].North 	:= fbENviroment.XpuTcIo(1).TileCoE(1,2).DiagData.TemperatureNorth;
	TileInfo[1].South 	:= fbENviroment.XpuTcIo(1).TileCoE(1,2).DiagData.TemperatureSouth;
	TileInfo[1].West 	:= fbENviroment.XpuTcIo(1).TileCoE(1,2).DiagData.TemperatureWest;
	TileInfo[1].FanRPM	:= fbENviroment.XpuTcIo(1).TileCoE(1,2).DiagData.FanRpm;
	
END_IF;
*)

(* SDO XPlanar APS diannosys data*)

slave_state(
	sNetId:='192.168.80.1.4.1',
	nSlaveAddr := 1001,
	bExecute := NOT slave_state.bBusy
);

IF NOT slave_state.bBusy THEN
	state := F_ConvSlaveStateToBits(slave_state.state);	
END_IF

// Get diganosis data from SDO
sdo_controller();
fbMqttPublish();

// Get diagnostics data every 0.5s
read_cycle_timer(IN := NOT read_cycle_timer.Q, PT := T#500MS);

IF read_cycle_timer.Q THEN
	sdo_controller.query(
					nSlaveAddr := 1001,
					bCompleteAccess := TRUE, 
					nIndex := 16#FA00, 
					nSubIndex := 0,
					pDstBuf := ADR(planar_tiles_diag_data[1]),
					cbBufLen := SIZEOF(planar_tiles_diag_data[1]),
					event_handler := fbMqttPublish
					);
	sdo_controller.query(
					nSlaveAddr := 1003,
					bCompleteAccess := TRUE, 
					nIndex := 16#FA00, 
					nSubIndex := 0,
					pDstBuf := ADR(planar_tiles_diag_data[2]),
					cbBufLen := SIZEOF(planar_tiles_diag_data[2]),
					event_handler := fbMqttPublish
					);
END_IF

// Database 
IF NOT db_initialize THEN
	fb_aps_diag_db_recorder.set_buffer_info(struct_size := SIZEOF(database_aps_diag_buffer[0]),
											buffer_size := SIZEOF(database_aps_diag_buffer),
											structure_name := 'ST_database_aps_diag');
	fb_aps_diag_db_recorder.SQL_parameters.table_name := 'xplanar_aps_diag';

	fb_mover_dynamics_recorder.set_buffer_info(struct_size := SIZEOF(database_mover_dynamics_buffer[0]),
											buffer_size := SIZEOF(database_mover_dynamics_buffer),
											structure_name := 'ST_mover_dynamics');
	fb_mover_dynamics_recorder.SQL_parameters.table_name := 'mover_dynamics';

	fb_ads_router_status_recorder.set_buffer_info(struct_size := SIZEOF(database_ads_router_info_buffer[0]),
											buffer_size := SIZEOF(database_ads_router_info_buffer),
											structure_name := 'ST_RouterStatusInfo');
	fb_ads_router_status_recorder.SQL_parameters.table_name := 'ADS_router_status';	
	fb_ads_router_status_recorder.max_chunk_size := 1;
	
	db_initialize := TRUE;
	fbMqttPublish.fbDatabaseRecorder REF= fb_aps_diag_db_recorder;
END_IF


